# B&R Automation Studio project TD52 (part 53)

```c
  /* BusSelector: '<S111>/Bus Selector12' */
  rtb_rSCR_NOxControlWaiting = UDC_B.BusInput1.rSCR_NOxControlWaiting;

  /* UnitDelay: '<S111>/Unit Delay' */
  rtb_UnitDelay = UDC_DWork.UnitDelay_DSTATE;

  /* BusSelector: '<S113>/Bus Selector1' */
  for (i = 0; i < 5; i++) {
    rtb_rUrClKiOffs_y[i] = UDC_B.BusInput2.CLNOx.rUrClKpOffs_x[i];
  }

  for (i = 0; i < 5; i++) {
    rtb_rUrClKiOffs_x[i] = UDC_B.BusInput2.CLNOx.rUrClKpOffs_y[i];
  }

  /* End of BusSelector: '<S113>/Bus Selector1' */
  /* Dynamic Look-Up Table Block: '<S113>/Lookup Table Dynamic'
   * Input0  Data Type:  Floating Point real32_T
   * Input1  Data Type:  Floating Point real32_T
   * Input2  Data Type:  Floating Point real32_T
   * Output0 Data Type:  Floating Point real32_T
   * Lookup Method: Linear_Endpoint
   *
   */
  LookUp_real32_T_real32_T( &(rtb_LookupTableDynamic1), rtb_rUrClKiOffs_x,
    rtb_Switch6, rtb_rUrClKiOffs_y, 4U, inst);

  /* Sum: '<S113>/Add2' */
  rtb_etaVolConst = rtb_LookupTableDynamic1 + UDC_B.BusInput1.rSCR_NOxCtrl_Kp;

  /* BusSelector: '<S111>/Bus Selector14' */
  rtb_bRel_SCR_Dosing_n = UDC_B.BusInput.bRel_SCR_Dosing;

  /* Logic: '<S111>/Logical Operator5' */
  rtb_RelationalOperator2 = (UDC_B.BusInput.bSCR_UreaDosingUnit_Man &&
    UDC_B.BusInput1.bSCR_UreaFlowCtrl_Active);

  /* Outputs for Atomic SubSystem: '<S111>/TON' */
  UDC_TON(rtb_bRel_SCR_Dosing_n, rtb_rSCR_NOxControlWaiting, &UDC_B.TON_f,
          &UDC_DWork.TON_f, inst);

  /* End of Outputs for SubSystem: '<S111>/TON' */

  /* Outputs for Atomic SubSystem: '<Root>/SlipDetection' */
  /* Logic: '<S111>/Logical Operator' incorporates:
   *  BusCreator: '<S10>/Bus Creator'
   *  Logic: '<S111>/Logical Operator3'
   */
  rtb_LogicalOperator_p = (UDC_B.BusInput2.CLNOx.bUrClRes ||
    rtb_RelationalOperator2 || (!UDC_B.TON_f.LogicalOperator3) ||
    UDC_B.BusInput.bSCR_Man || UDC_B.BusInput.bSCR_NOxControl_Man ||
    rtb_RelationalOperator_mq || UDC_B.BusInput.bSCR_NH3SlipDetect_Blocked);

  /* End of Outputs for SubSystem: '<Root>/SlipDetection' */

  /* Logic: '<S111>/Logical Operator8' incorporates:
   *  BusCreator: '<S9>/Bus Creator'
   */
  rtb_RelationalOperator2 = (rtb_bFreezeCtr_j || rtb_LogicalOperator_p);

  /* Switch: '<S111>/Switch1' incorporates:
   *  Constant: '<S111>/Constant'
   *  Gain: '<S111>/Gain'
   *  MATLAB Function: '<S119>/MATLAB Function'
   *  Sum: '<S111>/Add7'
   */
  if (rtb_RelationalOperator2) {
    rtb_LookupTableDynamic1 = 0.0F;
  } else {
    /* Outputs for Atomic SubSystem: '<S9>/E21_NOxCatOutManager' */
    rtb_LookupTableDynamic1 = -(rtb_BusCreator_h_rNOx_SCR_CatOu - rNOx_Act);

    /* End of Outputs for SubSystem: '<S9>/E21_NOxCatOutManager' */
  }

  /* End of Switch: '<S111>/Switch1' */

  /* Gain: '<S112>/Gain' */
  rtb_LookupTableDynamic1 *= 0.001F;

  /* Product: '<S112>/Product' */
  rtb_Product_f = rtb_etaVolConst * rtb_LookupTableDynamic1;

  /* DiscreteIntegrator: '<S112>/Discrete-Time Integrator' */
  if (UDC_DWork.DiscreteTimeIntegrator_IC_LOADI != 0) {
    UDC_DWork.DiscreteTimeIntegrator_DSTATE_p = UDC_B.BusInput2.CLNOx.rUrClI0;
    if (UDC_DWork.DiscreteTimeIntegrator_DSTATE_p >= 3.402823466E+38F) {
      UDC_DWork.DiscreteTimeIntegrator_DSTATE_p = 3.402823466E+38F;
    } else {
      if (UDC_DWork.DiscreteTimeIntegrator_DSTATE_p <= -3.402823466E+38F) {
        UDC_DWork.DiscreteTimeIntegrator_DSTATE_p = -3.402823466E+38F;
      }
    }
  }

  if (rtb_LogicalOperator_p || (UDC_DWork.DiscreteTimeIntegrator_PrevRe_j != 0))
  {
    UDC_DWork.DiscreteTimeIntegrator_DSTATE_p = UDC_B.BusInput2.CLNOx.rUrClI0;
    if (UDC_DWork.DiscreteTimeIntegrator_DSTATE_p >= 3.402823466E+38F) {
      UDC_DWork.DiscreteTimeIntegrator_DSTATE_p = 3.402823466E+38F;
    } else {
      if (UDC_DWork.DiscreteTimeIntegrator_DSTATE_p <= -3.402823466E+38F) {
        UDC_DWork.DiscreteTimeIntegrator_DSTATE_p = -3.402823466E+38F;
      }
    }
  }

  if (UDC_DWork.DiscreteTimeIntegrator_DSTATE_p >= 3.402823466E+38F) {
    UDC_DWork.DiscreteTimeIntegrator_DSTATE_p = 3.402823466E+38F;
  } else {
    if (UDC_DWork.DiscreteTimeIntegrator_DSTATE_p <= -3.402823466E+38F) {
      UDC_DWork.DiscreteTimeIntegrator_DSTATE_p = -3.402823466E+38F;
    }
  }

  rtb_DiscreteTimeIntegrator = UDC_DWork.DiscreteTimeIntegrator_DSTATE_p;

  /* End of DiscreteIntegrator: '<S112>/Discrete-Time Integrator' */

  /* BusSelector: '<S113>/Bus Selector4' */
  for (i = 0; i < 5; i++) {
    rtb_rUrClKiOffs_x[i] = UDC_B.BusInput2.CLNOx.rUrClKdOffs_x[i];
  }

  for (i = 0; i < 5; i++) {
    rtb_rUrClKiOffs_y[i] = UDC_B.BusInput2.CLNOx.rUrClKdOffs_y[i];
  }

  /* End of BusSelector: '<S113>/Bus Selector4' */
  /* Dynamic Look-Up Table Block: '<S113>/Lookup Table Dynamic2'
   * Input0  Data Type:  Floating Point real32_T
   * Input1  Data Type:  Floating Point real32_T
   * Input2  Data Type:  Floating Point real32_T
   * Output0 Data Type:  Floating Point real32_T
   * Lookup Method: Linear_Endpoint
   *
   */
  LookUp_real32_T_real32_T( &(rtb_Switch2_mg), rtb_rUrClKiOffs_y, rtb_Switch6,
    rtb_rUrClKiOffs_x, 4U, inst);

  /* Product: '<S112>/Product2' incorporates:
   *  Sum: '<S113>/Add3'
   */
  rtb_etaVolConst = (rtb_Switch2_mg + UDC_B.BusInput1.rSCR_NOxCtrl_Kd) *
    rtb_LookupTableDynamic1;

  /* DiscreteIntegrator: '<S112>/Discrete-Time Integrator1' */
  if (UDC_DWork.DiscreteTimeIntegrator1_IC_LOAD != 0) {
    UDC_DWork.DiscreteTimeIntegrator1_DSTATE = UDC_B.BusInput2.CLNOx.rUrClD0;
    if (UDC_DWork.DiscreteTimeIntegrator1_DSTATE >= 3.402823466E+38F) {
      UDC_DWork.DiscreteTimeIntegrator1_DSTATE = 3.402823466E+38F;
    } else {
      if (UDC_DWork.DiscreteTimeIntegrator1_DSTATE <= -3.402823466E+38F) {
        UDC_DWork.DiscreteTimeIntegrator1_DSTATE = -3.402823466E+38F;
      }
    }
  }

  if (rtb_LogicalOperator_p || (UDC_DWork.DiscreteTimeIntegrator1_PrevRes != 0))
  {
    UDC_DWork.DiscreteTimeIntegrator1_DSTATE = UDC_B.BusInput2.CLNOx.rUrClD0;
    if (UDC_DWork.DiscreteTimeIntegrator1_DSTATE >= 3.402823466E+38F) {
      UDC_DWork.DiscreteTimeIntegrator1_DSTATE = 3.402823466E+38F;
    } else {
      if (UDC_DWork.DiscreteTimeIntegrator1_DSTATE <= -3.402823466E+38F) {
        UDC_DWork.DiscreteTimeIntegrator1_DSTATE = -3.402823466E+38F;
      }
    }
  }

  if (UDC_DWork.DiscreteTimeIntegrator1_DSTATE >= 3.402823466E+38F) {
    UDC_DWork.DiscreteTimeIntegrator1_DSTATE = 3.402823466E+38F;
  } else {
    if (UDC_DWork.DiscreteTimeIntegrator1_DSTATE <= -3.402823466E+38F) {
      UDC_DWork.DiscreteTimeIntegrator1_DSTATE = -3.402823466E+38F;
    }
  }

  rtb_Switch2_mg = UDC_DWork.DiscreteTimeIntegrator1_DSTATE;

  /* End of DiscreteIntegrator: '<S112>/Discrete-Time Integrator1' */

  /* Product: '<S112>/Product3' incorporates:
   *  Sum: '<S112>/Sum2'
   */
  rtb_Product3 = (rtb_etaVolConst - rtb_Switch2_mg) *
    UDC_B.BusInput2.CLNOx.rUrClN;

  /* Switch: '<S111>/Switch' incorporates:
   *  BusCreator: '<S9>/Bus Creator'
   *  Sum: '<S112>/Sum1'
   */
  if (!rtb_bFreezeCtr_j) {
    rtb_UnitDelay = (rtb_Product_f + rtb_DiscreteTimeIntegrator) + rtb_Product3;
  }

  /* End of Switch: '<S111>/Switch' */

  /* Switch: '<S114>/Switch2' incorporates:
   *  RelationalOperator: '<S114>/LowerRelop1'
   *  RelationalOperator: '<S114>/UpperRelop'
   *  Switch: '<S114>/Switch'
   */
  if (rtb_UnitDelay > UDC_B.BusInput1.rSCR_NOxCtrl_Ymax) {
    rtb_Switch2_m = UDC_B.BusInput1.rSCR_NOxCtrl_Ymax;
  } else if (rtb_UnitDelay < UDC_B.BusInput1.rSCR_NOxCtrl_Ymin) {
    /* Switch: '<S114>/Switch' */
    rtb_Switch2_m = UDC_B.BusInput1.rSCR_NOxCtrl_Ymin;
  } else {
    rtb_Switch2_m = rtb_UnitDelay;
  }

  /* End of Switch: '<S114>/Switch2' */

  /* Switch: '<S8>/Switch1' incorporates:
   *  Constant: '<S8>/const1'
   *  Switch: '<S8>/Switch7'
   */
  if (UDC_B.BusInput.bSCR_NOxControl_Man) {
    rtb_Switch_ah = UDC_B.BusInput.rFlow_SCR_UreaDosingUnit_spMan;
  } else if (UDC_B.BusInput.bRel_SCR_Dosing) {
    /* Switch: '<S8>/Switch7' incorporates:
     *  Sum: '<S8>/Add6'
     */
    rtb_Switch_ah = rtb_rFlow_SCR_UreaDosing_ffNH3C + rtb_Switch2_m;
  } else {
    rtb_Switch_ah = 0.0F;
  }

  /* End of Switch: '<S8>/Switch1' */

  /* Switch: '<S110>/Switch2' incorporates:
   *  Constant: '<S8>/const2'
   *  RelationalOperator: '<S110>/LowerRelop1'
   *  RelationalOperator: '<S110>/UpperRelop'
   *  Switch: '<S110>/Switch'
   */
  if (rtb_Switch_ah > UDC_B.BusInput1.rFlow_SCR_UreaDosingUnit_Hi) {
    rtb_Switch2_h = UDC_B.BusInput1.rFlow_SCR_UreaDosingUnit_Hi;
  } else if (rtb_Switch_ah < 0.0F) {
    /* Switch: '<S110>/Switch' incorporates:
     *  Constant: '<S8>/const2'
     */
    rtb_Switch2_h = 0.0F;
  } else {
    rtb_Switch2_h = rtb_Switch_ah;
  }

  /* End of Switch: '<S110>/Switch2' */

  /* If: '<S6>/If' incorporates:
   *  Constant: '<S84>/Constant'
   *  Constant: '<S84>/Constant1'
   *  Constant: '<S84>/Constant2'
   *  Constant: '<S84>/Constant7'
   *  Constant: '<S84>/Constant8'
   */
  if (UDC_B.BusInput1.bSCR_UreaDosingValve_Exist &&
      UDC_B.BusInput1.bSCR_UreaFlowCtrl_Active) {
    /* Outputs for IfAction SubSystem: '<S6>/UrValCntr' incorporates:
     *  ActionPort: '<S86>/Action Port'
     */
    /* Sum: '<S86>/Add2' */
    rtb_etaVolConst = UDC_B.BusInput2.CLVal.rUrValKpOffs +
      UDC_B.BusInput1.rSCR_UreaFlowCtrl_Kp;

    /* Switch: '<S86>/Switch1' incorporates:
     *  Constant: '<S86>/Constant'
     *  Sum: '<S86>/Add7'
     */
    if (UDC_B.BusInput.tFlow_SCR_UreaDosingOut.GoodQual) {
      rtb_Product_k = rtb_Switch2_h - UDC_B.BusInput.tFlow_SCR_UreaDosingOut.Ai;
    } else {
      rtb_Product_k = 0.0F;
    }

    /* End of Switch: '<S86>/Switch1' */

    /* Gain: '<S94>/Gain' */
    rtb_sampletime_c = 0.01F * rtb_Product_k;

    /* Product: '<S94>/Product' */
    rtb_Product_k = rtb_etaVolConst * rtb_sampletime_c;

    /* Logic: '<S86>/Logical Operator' incorporates:
     *  Logic: '<S86>/Logical Operator1'
     *  Logic: '<S86>/Logical Operator2'
     *  Logic: '<S86>/Logical Operator3'
     */
    rtb_LogicalOperator_g = (UDC_B.BusInput2.CLVal.bUrValRes ||
      (!UDC_B.BusInput1.bSCR_UreaDosingValve_Exist) ||
      (!UDC_B.BusInput.bRel_SCR_Dosing) ||
      (!UDC_B.BusInput1.bSCR_UreaFlowCtrl_Active) || UDC_B.BusInput.bSCR_Man ||
      UDC_B.BusInput.bSCR_UreaDosingUnit_Man);

    /* DiscreteIntegrator: '<S94>/Discrete-Time Integrator' */
    if (UDC_DWork.DiscreteTimeIntegrator_IC_LOA_f != 0) {
      UDC_DWork.DiscreteTimeIntegrator_DSTATE_e = UDC_B.BusInput2.CLVal.rUrValI0;
      if (UDC_DWork.DiscreteTimeIntegrator_DSTATE_e >= 3.402823466E+38F) {
        UDC_DWork.DiscreteTimeIntegrator_DSTATE_e = 3.402823466E+38F;
      } else {
        if (UDC_DWork.DiscreteTimeIntegrator_DSTATE_e <= -3.402823466E+38F) {
          UDC_DWork.DiscreteTimeIntegrator_DSTATE_e = -3.402823466E+38F;
        }
      }
    }

    if (rtb_LogicalOperator_g || (UDC_DWork.DiscreteTimeIntegrator_PrevRe_p != 0))
    {
      UDC_DWork.DiscreteTimeIntegrator_DSTATE_e = UDC_B.BusInput2.CLVal.rUrValI0;
      if (UDC_DWork.DiscreteTimeIntegrator_DSTATE_e >= 3.402823466E+38F) {
        UDC_DWork.DiscreteTimeIntegrator_DSTATE_e = 3.402823466E+38F;
      } else {
        if (UDC_DWork.DiscreteTimeIntegrator_DSTATE_e <= -3.402823466E+38F) {
          UDC_DWork.DiscreteTimeIntegrator_DSTATE_e = -3.402823466E+38F;
        }
      }
    }

    if (UDC_DWork.DiscreteTimeIntegrator_DSTATE_e >= 3.402823466E+38F) {
      UDC_DWork.DiscreteTimeIntegrator_DSTATE_e = 3.402823466E+38F;
    } else {
      if (UDC_DWork.DiscreteTimeIntegrator_DSTATE_e <= -3.402823466E+38F) {
        UDC_DWork.DiscreteTimeIntegrator_DSTATE_e = -3.402823466E+38F;
      }
    }

    rtb_DiscreteTimeIntegrator_p = UDC_DWork.DiscreteTimeIntegrator_DSTATE_e;

    /* Sum: '<S86>/Add6' */
    rtb_etaVolConst = UDC_B.BusInput2.CLVal.rUrValKdOffs +
      UDC_B.BusInput1.rSCR_UreaFlowCtrl_Kd;

    /* DiscreteIntegrator: '<S94>/Discrete-Time Integrator1' */
    if (UDC_DWork.DiscreteTimeIntegrator1_IC_LO_i != 0) {
      UDC_DWork.DiscreteTimeIntegrator1_DSTAT_b = UDC_B.BusInput2.CLVal.rUrValD0;
      if (UDC_DWork.DiscreteTimeIntegrator1_DSTAT_b >= 3.402823466E+38F) {
        UDC_DWork.DiscreteTimeIntegrator1_DSTAT_b = 3.402823466E+38F;
      } else {
        if (UDC_DWork.DiscreteTimeIntegrator1_DSTAT_b <= -3.402823466E+38F) {
          UDC_DWork.DiscreteTimeIntegrator1_DSTAT_b = -3.402823466E+38F;
        }
      }
    }

    if (rtb_LogicalOperator_g || (UDC_DWork.DiscreteTimeIntegrator1_PrevR_e != 0))
    {
      UDC_DWork.DiscreteTimeIntegrator1_DSTAT_b = UDC_B.BusInput2.CLVal.rUrValD0;
      if (UDC_DWork.DiscreteTimeIntegrator1_DSTAT_b >= 3.402823466E+38F) {
        UDC_DWork.DiscreteTimeIntegrator1_DSTAT_b = 3.402823466E+38F;
      } else {
        if (UDC_DWork.DiscreteTimeIntegrator1_DSTAT_b <= -3.402823466E+38F) {
          UDC_DWork.DiscreteTimeIntegrator1_DSTAT_b = -3.402823466E+38F;
        }
      }
    }

    if (UDC_DWork.DiscreteTimeIntegrator1_DSTAT_b >= 3.402823466E+38F) {
      UDC_DWork.DiscreteTimeIntegrator1_DSTAT_b = 3.402823466E+38F;
    } else {
      if (UDC_DWork.DiscreteTimeIntegrator1_DSTAT_b <= -3.402823466E+38F) {
        UDC_DWork.DiscreteTimeIntegrator1_DSTAT_b = -3.402823466E+38F;
      }
    }

    /* Product: '<S94>/Product3' incorporates:
     *  DiscreteIntegrator: '<S94>/Discrete-Time Integrator1'
     *  Product: '<S94>/Product2'
     *  Sum: '<S94>/Sum2'
     */
    rtb_Product3_i = (rtb_etaVolConst * rtb_sampletime_c -
                      UDC_DWork.DiscreteTimeIntegrator1_DSTAT_b) *
      UDC_B.BusInput2.CLVal.rUrValN;

    /* Switch: '<S86>/Switch' incorporates:
     *  DiscreteIntegrator: '<S94>/Discrete-Time Integrator'
     *  Sum: '<S94>/Sum1'
     *  UnitDelay: '<S86>/Unit Delay'
     */
    if (UDC_B.BusInput.tFlow_SCR_UreaDosingOut.GoodQual) {
      rtb_Switch2_kp = (rtb_Product_k +
                        UDC_DWork.DiscreteTimeIntegrator_DSTATE_e) +
        rtb_Product3_i;
    } else {
      rtb_Switch2_kp = UDC_DWork.UnitDelay_DSTATE_n;
    }

    /* End of Switch: '<S86>/Switch' */

    /* Switch: '<S95>/Switch2' incorporates:
     *  RelationalOperator: '<S95>/LowerRelop1'
     *  RelationalOperator: '<S95>/UpperRelop'
     *  Switch: '<S95>/Switch'
     */
    if (rtb_Switch2_kp > UDC_B.BusInput1.rSCR_UreaFlowCtrl_Ymax) {
      rtb_Switch2_p = UDC_B.BusInput1.rSCR_UreaFlowCtrl_Ymax;
    } else if (rtb_Switch2_kp < UDC_B.BusInput1.rSCR_UreaFlowCtrl_Ymin) {
      /* Switch: '<S95>/Switch' */
      rtb_Switch2_p = UDC_B.BusInput1.rSCR_UreaFlowCtrl_Ymin;
    } else {
      rtb_Switch2_p = rtb_Switch2_kp;
    }

    /* End of Switch: '<S95>/Switch2' */

    /* Abs: '<S93>/Abs' incorporates:
     *  BusSelector: '<S86>/Bus Selector1'
     */
    rtb_LookupTableDynamic_e = (real32_T)fabs
      (UDC_B.BusInput1.rFlow_SCR_UreaDosingValveCoeff);

    /* Switch: '<S93>/Switch' incorporates:
     *  BusSelector: '<S86>/Bus Selector1'
     *  Constant: '<S93>/Constant2'
     *  RelationalOperator: '<S93>/Relational Operator'
     */
    if (1.1920929E-7F >= rtb_LookupTableDynamic_e) {
      rtb_Switch_f = 1.1920929E-7F;
    } else {
      rtb_Switch_f = UDC_B.BusInput1.rFlow_SCR_UreaDosingValveCoeff;
    }

    /* End of Switch: '<S93>/Switch' */

    /* UnitDelay: '<S97>/Unit Delay' */
    rtb_LookupTableDynamic_e = UDC_DWork.UnitDelay_DSTATE_d;

    /* Switch: '<S97>/Switch' */
    if (UDC_B.BusInput.tDPr_UreaDosingUnit.GoodQual) {
      rtb_Switch_ld = UDC_B.BusInput.tDPr_UreaDosingUnit.Ai;
    } else {
      rtb_Switch_ld = rtb_LookupTableDynamic_e;
    }

    /* End of Switch: '<S97>/Switch' */

    /* BusSelector: '<S97>/Bus Selector2' */
    for (i = 0; i < 11; i++) {
      rtb_rUrValLinMap_x[i] = UDC_B.BusInput2.CLVal.rUrValLinMap_x[i];
    }

    for (i = 0; i < 11; i++) {
      rtb_rUrValLinMap_y[i] = UDC_B.BusInput2.CLVal.rUrValLinMap_y[i];
    }

    rtb_rTiFilt_DPrVlv = UDC_B.BusInput2.CLVal.rTiFilt_DPrVlv;

    /* End of BusSelector: '<S97>/Bus Selector2' */

    /* Outputs for Atomic SubSystem: '<S97>/Filter_DPr' */
    UDC_Filter(rtb_rTiFilt_DPrVlv, rtb_LogicalOperator_g, rtb_Switch_ld,
               &UDC_B.Filter_DPr, &UDC_DWork.Filter_DPr, inst);

    /* End of Outputs for SubSystem: '<S97>/Filter_DPr' */

    /* Product: '<S97>/Divide2' incorporates:
     *  Gain: '<S97>/Gain'
     */
    rtb_LookupTableDynamic_e = UDC_B.Filter_DPr.Switch / (0.001F * rtb_Switch);

    /* Saturate: '<S97>/Saturation' */
    if (rtb_LookupTableDynamic_e >= 1.0E+6F) {
      rtb_LookupTableDynamic_e = 1.0E+6F;
    } else {
      if (rtb_LookupTableDynamic_e <= 0.001F) {
        rtb_LookupTableDynamic_e = 0.001F;
      }
    }

    /* End of Saturate: '<S97>/Saturation' */

    /* Sqrt: '<S97>/Sqrt' */
    rtb_LookupTableDynamic_e = (real32_T)sqrt(rtb_LookupTableDynamic_e);

    /* Abs: '<S100>/Abs' */
    rtb_Switch_h = (real32_T)fabs(rtb_LookupTableDynamic_e);

    /* Switch: '<S100>/Switch' incorporates:
     *  Constant: '<S100>/Constant2'
     *  RelationalOperator: '<S100>/Relational Operator'
     */
    if (1.1920929E-7F >= rtb_Switch_h) {
      rtb_LookupTableDynamic_e = 1.1920929E-7F;
    }

    /* End of Switch: '<S100>/Switch' */

    /* Product: '<S97>/Divide1' */
    rtb_LookupTableDynamic_e = rtb_Switch2_h / rtb_Switch_f /
      rtb_LookupTableDynamic_e;

    /* Dynamic Look-Up Table Block: '<S97>/Lookup Table Dynamic'
     * Input0  Data Type:  Floating Point real32_T
     * Input1  Data Type:  Floating Point real32_T
     * Input2  Data Type:  Floating Point real32_T
     * Output0 Data Type:  Floating Point real32_T
     * Lookup Method: Linear_Endpoint
     *
     */
    LookUp_real32_T_real32_T( &(rtb_Switch_h), rtb_rUrValLinMap_y,
      rtb_LookupTableDynamic_e, rtb_rUrValLinMap_x, 10U, inst);

    /* Sum: '<S86>/Add3' */
    rtb_LookupTableDynamic_e = rtb_Switch_h + rtb_Switch2_p;

    /* Product: '<S86>/Divide1' incorporates:
     *  Sum: '<S86>/Add1'
     */
    rtb_etaVolConst = (rtb_Switch2_kp - rtb_Switch2_p) *
      UDC_B.BusInput2.CLVal.rUrValKaw;

    /* Product: '<S86>/Divide6' incorporates:
     *  Sum: '<S86>/Add10'
     */
    rtb_Gain1 = (rtb_LookupTableDynamic_e -
                 UDC_B.BusInput.rPos_SCR_UreaDosingValve) *
      UDC_B.BusInput2.CLVal.rUrValKawExt;

    /* Saturate: '<S86>/Saturation1' */
    if (rtb_LookupTableDynamic_e >= 1.0F) {
      rtb_Saturation1_f = 1.0F;
    } else if (rtb_LookupTableDynamic_e <= 0.0F) {
      rtb_Saturation1_f = 0.0F;
    } else {
      rtb_Saturation1_f = rtb_LookupTableDynamic_e;
    }

    /* End of Saturate: '<S86>/Saturation1' */

    /* Product: '<S86>/Divide2' incorporates:
     *  Sum: '<S86>/Add8'
     */
    rtb_UkYk1 = (rtb_LookupTableDynamic_e - rtb_Saturation1_f) *
      UDC_B.BusInput2.CLVal.rUrValKaw;

    /* Sum: '<S86>/Add4' */
    rtb_etaVolConst = (rtb_etaVolConst + rtb_Gain1) + rtb_UkYk1;

    /* Sum: '<S86>/Add5' */
    rtb_UkYk1 = UDC_B.BusInput2.CLVal.rUrValKiOffs +
      UDC_B.BusInput1.rSCR_UreaFlowCtrl_Ki;

    /* Switch: '<S96>/Switch2' incorporates:
     *  Gain: '<S86>/Gain3'
     *  RelationalOperator: '<S96>/LowerRelop1'
     *  RelationalOperator: '<S96>/UpperRelop'
     *  Switch: '<S96>/Switch'
     */
    if (rtb_etaVolConst > UDC_B.BusInput1.rFlow_SCR_UreaDosingUnit_Hi) {
      rtb_LookupTableDynamic_e = UDC_B.BusInput1.rFlow_SCR_UreaDosingUnit_Hi;
    } else if (rtb_etaVolConst < -UDC_B.BusInput1.rFlow_SCR_UreaDosingUnit_Hi) {
      /* Switch: '<S96>/Switch' incorporates:
       *  Gain: '<S86>/Gain3'
       */
      rtb_LookupTableDynamic_e = -UDC_B.BusInput1.rFlow_SCR_UreaDosingUnit_Hi;
    } else {
      /* Switch: '<S96>/Switch' */
      rtb_LookupTableDynamic_e = rtb_etaVolConst;
    }

    /* End of Switch: '<S96>/Switch2' */

    /* Gain: '<S86>/Gain2' */
    rtb_LookupTableDynamic_e = -rtb_LookupTableDynamic_e;

    /* Logic: '<S86>/Logical Operator4' */
    rtb_LogicalOperator1_b = !rtb_LogicalOperator_g;

    /* Sum: '<S94>/Add' */
    rtb_etaVolConst = rtb_sampletime_c + rtb_LookupTableDynamic_e;

    /* BusCreator: '<S94>/Bus Creator' */
    rtb_sampletime_c = rtb_LookupTableDynamic_e;

    /* SignalConversion: '<S86>/Signal Conversion' */
    UDC_B.Merge5[0] = rtb_Switch_h;

    /* SignalConversion: '<S86>/Signal Conversion1' */
    UDC_B.Merge5[1] = rtb_Saturation1_f;

    /* SignalConversion: '<S86>/Signal Conversion2' */
    UDC_B.Merge5[2] = rtb_Switch2_p;

    /* BusSelector: '<S98>/Bus Selector4' */
    for (i = 0; i < 11; i++) {
      rtb_rUrValLinMap_y[i] = UDC_B.BusInput2.CLVal.rUrValLinMap_y[i];
    }

    for (i = 0; i < 11; i++) {
      rtb_rUrValLinMap_x[i] = UDC_B.BusInput2.CLVal.rUrValLinMap_x[i];
    }

    rtb_rTiFilt_DPrVlv_b = UDC_B.BusInput2.CLVal.rTiFilt_DPrVlv;

    /* End of BusSelector: '<S98>/Bus Selector4' */

    /* UnitDelay: '<S98>/Unit Delay2' */
    rtb_Switch_h = UDC_DWork.UnitDelay2_DSTATE;

    /* Switch: '<S98>/Switch3' */
    if (UDC_B.BusInput.tDPr_UreaDosingUnit.GoodQual) {
      rtb_Switch3_l = UDC_B.BusInput.tDPr_UreaDosingUnit.Ai;
    } else {
      rtb_Switch3_l = rtb_Switch_h;
    }

    /* End of Switch: '<S98>/Switch3' */

    /* Outputs for Atomic SubSystem: '<S98>/Filter_DPr' */
    UDC_Filter(rtb_rTiFilt_DPrVlv_b, rtb_LogicalOperator_g, rtb_Switch3_l,
               &UDC_B.Filter_DPr_h, &UDC_DWork.Filter_DPr_h, inst);

    /* End of Outputs for SubSystem: '<S98>/Filter_DPr' */

    /* Product: '<S98>/Divide5' incorporates:
     *  Gain: '<S98>/Gain1'
     */
    rtb_Switch_h = UDC_B.Filter_DPr_h.Switch / (0.001F * rtb_Switch);

    /* Saturate: '<S98>/Saturation2' */
    if (rtb_Switch_h >= 1.0E+6F) {
      rtb_Switch_h = 1.0E+6F;
    } else {
      if (rtb_Switch_h <= 0.001F) {
        rtb_Switch_h = 0.001F;
      }
    }

    /* End of Saturate: '<S98>/Saturation2' */

    /* Sqrt: '<S98>/Sqrt1' */
    rtb_Switch_h = (real32_T)sqrt(rtb_Switch_h);

    /* Abs: '<S105>/Abs' */
    rtb_LookupTableDynamic_e = (real32_T)fabs(rtb_Switch_h);

    /* Switch: '<S105>/Switch' incorporates:
     *  Constant: '<S105>/Constant2'
     *  RelationalOperator: '<S105>/Relational Operator'
     */
    if (1.1920929E-7F >= rtb_LookupTableDynamic_e) {
      rtb_Switch_h = 1.1920929E-7F;
    }

    /* End of Switch: '<S105>/Switch' */
    /* Dynamic Look-Up Table Block: '<S98>/Lookup Table Dynamic'
     * Input0  Data Type:  Floating Point real32_T
     * Input1  Data Type:  Floating Point real32_T
     * Input2  Data Type:  Floating Point real32_T
     * Output0 Data Type:  Floating Point real32_T
     * Lookup Method: Linear_Endpoint
     *
     */
    LookUp_real32_T_real32_T( &(rtb_LookupTableDynamic_e), rtb_rUrValLinMap_x,
      rtb_Saturation1_f, rtb_rUrValLinMap_y, 10U, inst);

    /* Product: '<S98>/Divide4' */
    UDC_B.Merge5[3] = rtb_Switch_h * rtb_Switch_f * rtb_LookupTableDynamic_e;

    /* Update for DiscreteIntegrator: '<S94>/Discrete-Time Integrator' incorporates:
     *  Product: '<S94>/Product1'
     */
    UDC_DWork.DiscreteTimeIntegrator_IC_LOA_f = 0U;
    if (!rtb_LogicalOperator_g) {
      UDC_DWork.DiscreteTimeIntegrator_DSTATE_e += rtb_UkYk1 * rtb_etaVolConst *
        0.1F;
      if (UDC_DWork.DiscreteTimeIntegrator_DSTATE_e >= 3.402823466E+38F) {
        UDC_DWork.DiscreteTimeIntegrator_DSTATE_e = 3.402823466E+38F;
      } else {
        if (UDC_DWork.DiscreteTimeIntegrator_DSTATE_e <= -3.402823466E+38F) {
          UDC_DWork.DiscreteTimeIntegrator_DSTATE_e = -3.402823466E+38F;
        }
      }
    }

    if (rtb_LogicalOperator_g) {
      UDC_DWork.DiscreteTimeIntegrator_PrevRe_p = 1;
    } else {
      UDC_DWork.DiscreteTimeIntegrator_PrevRe_p = 0;
    }

    /* End of Update for DiscreteIntegrator: '<S94>/Discrete-Time Integrator' */

    /* Update for DiscreteIntegrator: '<S94>/Discrete-Time Integrator1' */
    UDC_DWork.DiscreteTimeIntegrator1_IC_LO_i = 0U;
    if (!rtb_LogicalOperator_g) {
      UDC_DWork.DiscreteTimeIntegrator1_DSTAT_b += 0.1F * rtb_Product3_i;
      if (UDC_DWork.DiscreteTimeIntegrator1_DSTAT_b >= 3.402823466E+38F) {
        UDC_DWork.DiscreteTimeIntegrator1_DSTAT_b = 3.402823466E+38F;
      } else {
        if (UDC_DWork.DiscreteTimeIntegrator1_DSTAT_b <= -3.402823466E+38F) {
          UDC_DWork.DiscreteTimeIntegrator1_DSTAT_b = -3.402823466E+38F;
        }
      }
    }

    if (rtb_LogicalOperator_g) {
      UDC_DWork.DiscreteTimeIntegrator1_PrevR_e = 1;
    } else {
      UDC_DWork.DiscreteTimeIntegrator1_PrevR_e = 0;
    }

    /* End of Update for DiscreteIntegrator: '<S94>/Discrete-Time Integrator1' */

    /* Update for UnitDelay: '<S86>/Unit Delay' */
    UDC_DWork.UnitDelay_DSTATE_n = rtb_Switch2_kp;

    /* Update for UnitDelay: '<S97>/Unit Delay' */
    UDC_DWork.UnitDelay_DSTATE_d = rtb_Switch_ld;

    /* Update for UnitDelay: '<S98>/Unit Delay2' */
    UDC_DWork.UnitDelay2_DSTATE = rtb_Switch3_l;

    /* End of Outputs for SubSystem: '<S6>/UrValCntr' */
  } else if (UDC_B.BusInput1.bSCR_UreaFlowCtrl_Active) {
    /* Outputs for IfAction SubSystem: '<S6>/UrPumpCntr' incorporates:
     *  ActionPort: '<S85>/Action Port'
     */
    /* BusSelector: '<S85>/Bus Selector2' */
    for (i = 0; i < 11; i++) {
      rtb_rUrPpCntrFFMap_x[i] = UDC_B.BusInput2.CLPp.rUrPpCntrFFMap_x[i];
    }

    for (i = 0; i < 11; i++) {
      rtb_rUrPpCntrFFMap_y[i] = UDC_B.BusInput2.CLPp.rUrPpCntrFFMap_y[i];
    }

    /* End of BusSelector: '<S85>/Bus Selector2' */

    /* Sum: '<S85>/Add2' */
    rtb_etaVolConst = UDC_B.BusInput2.CLPp.rUrPpKpOffs +
      UDC_B.BusInput1.rSCR_UreaFlowCtrl_Kp;

    /* Switch: '<S85>/Switch1' incorporates:
     *  Constant: '<S85>/Constant'
     *  Logic: '<S85>/Logical Operator6'
     *  Sum: '<S85>/Add7'
     */
    if (UDC_B.BusInput.tFlow_SCR_UreaDosingOut.GoodQual &&
        UDC_B.BusInput1.bFlow_SCR_UreaDosingOut_Exist) {
      rtb_Product_k = rtb_Switch2_h - UDC_B.BusInput.tFlow_SCR_UreaDosingOut.Ai;
    } else {
      rtb_Product_k = 0.0F;
    }

    /* End of Switch: '<S85>/Switch1' */

    /* Gain: '<S88>/Gain' */
    rtb_sampletime_c = 0.01F * rtb_Product_k;

    /* Product: '<S88>/Product' */
    rtb_Product_k = rtb_etaVolConst * rtb_sampletime_c;

    /* Logic: '<S85>/Logical Operator2' incorporates:
     *  Logic: '<S85>/Logical Operator1'
     *  Logic: '<S85>/Logical Operator3'
     *  Logic: '<S85>/Logical Operator5'
     */
    rtb_LogicalOperator2_j = (UDC_B.BusInput2.CLPp.bUrPpRes ||
      (!UDC_B.BusInput1.bSCR_UreaFlowCtrl_Active) ||
      (!UDC_B.BusInput.bRel_SCR_Dosing) || UDC_B.BusInput.bSCR_Man ||
      UDC_B.BusInput.bSCR_UreaDosingUnit_Man ||
      (!UDC_B.BusInput1.bFlow_SCR_UreaDosingOut_Exist));

    /* DiscreteIntegrator: '<S88>/Discrete-Time Integrator' */
    if (UDC_DWork.DiscreteTimeIntegrator_IC_LOA_e != 0) {
      UDC_DWork.DiscreteTimeIntegrator_DSTATE_d = UDC_B.BusInput2.CLPp.rUrPpI0;
      if (UDC_DWork.DiscreteTimeIntegrator_DSTATE_d >= 3.402823466E+38F) {
        UDC_DWork.DiscreteTimeIntegrator_DSTATE_d = 3.402823466E+38F;
      } else {
        if (UDC_DWork.DiscreteTimeIntegrator_DSTATE_d <= -3.402823466E+38F) {
          UDC_DWork.DiscreteTimeIntegrator_DSTATE_d = -3.402823466E+38F;
        }
      }
    }

    if (rtb_LogicalOperator2_j || (UDC_DWork.DiscreteTimeIntegrator_PrevR_j5 !=
         0)) {
      UDC_DWork.DiscreteTimeIntegrator_DSTATE_d = UDC_B.BusInput2.CLPp.rUrPpI0;
      if (UDC_DWork.DiscreteTimeIntegrator_DSTATE_d >= 3.402823466E+38F) {
        UDC_DWork.DiscreteTimeIntegrator_DSTATE_d = 3.402823466E+38F;
      } else {
        if (UDC_DWork.DiscreteTimeIntegrator_DSTATE_d <= -3.402823466E+38F) {
          UDC_DWork.DiscreteTimeIntegrator_DSTATE_d = -3.402823466E+38F;
        }
      }
    }

    if (UDC_DWork.DiscreteTimeIntegrator_DSTATE_d >= 3.402823466E+38F) {
      UDC_DWork.DiscreteTimeIntegrator_DSTATE_d = 3.402823466E+38F;
    } else {
      if (UDC_DWork.DiscreteTimeIntegrator_DSTATE_d <= -3.402823466E+38F) {
        UDC_DWork.DiscreteTimeIntegrator_DSTATE_d = -3.402823466E+38F;
      }
    }

    rtb_DiscreteTimeIntegrator_p = UDC_DWork.DiscreteTimeIntegrator_DSTATE_d;

    /* Sum: '<S85>/Add6' */
    rtb_etaVolConst = UDC_B.BusInput2.CLPp.rUrPpKdOffs +
      UDC_B.BusInput1.rSCR_UreaFlowCtrl_Kd;

    /* DiscreteIntegrator: '<S88>/Discrete-Time Integrator1' */
    if (UDC_DWork.DiscreteTimeIntegrator1_IC_LO_n != 0) {
      UDC_DWork.DiscreteTimeIntegrator1_DSTAT_l = UDC_B.BusInput2.CLPp.rUrPpD0;
      if (UDC_DWork.DiscreteTimeIntegrator1_DSTAT_l >= 3.402823466E+38F) {
        UDC_DWork.DiscreteTimeIntegrator1_DSTAT_l = 3.402823466E+38F;
      } else {
        if (UDC_DWork.DiscreteTimeIntegrator1_DSTAT_l <= -3.402823466E+38F) {
          UDC_DWork.DiscreteTimeIntegrator1_DSTAT_l = -3.402823466E+38F;
        }
      }
    }

    if (rtb_LogicalOperator2_j || (UDC_DWork.DiscreteTimeIntegrator1_PrevR_b !=
         0)) {
      UDC_DWork.DiscreteTimeIntegrator1_DSTAT_l = UDC_B.BusInput2.CLPp.rUrPpD0;
      if (UDC_DWork.DiscreteTimeIntegrator1_DSTAT_l >= 3.402823466E+38F) {
        UDC_DWork.DiscreteTimeIntegrator1_DSTAT_l = 3.402823466E+38F;
      } else {
        if (UDC_DWork.DiscreteTimeIntegrator1_DSTAT_l <= -3.402823466E+38F) {
          UDC_DWork.DiscreteTimeIntegrator1_DSTAT_l = -3.402823466E+38F;
        }
      }
    }

    if (UDC_DWork.DiscreteTimeIntegrator1_DSTAT_l >= 3.402823466E+38F) {
      UDC_DWork.DiscreteTimeIntegrator1_DSTAT_l = 3.402823466E+38F;
    } else {
      if (UDC_DWork.DiscreteTimeIntegrator1_DSTAT_l <= -3.402823466E+38F) {
        UDC_DWork.DiscreteTimeIntegrator1_DSTAT_l = -3.402823466E+38F;
      }
    }

    /* Product: '<S88>/Product3' incorporates:
     *  DiscreteIntegrator: '<S88>/Discrete-Time Integrator1'
     *  Product: '<S88>/Product2'
     *  Sum: '<S88>/Sum2'
     */
    rtb_Product3_i = (rtb_etaVolConst * rtb_sampletime_c -
                      UDC_DWork.DiscreteTimeIntegrator1_DSTAT_l) *
      UDC_B.BusInput2.CLPp.rUrPpN;

    /* Switch: '<S85>/Switch' incorporates:
     *  DiscreteIntegrator: '<S88>/Discrete-Time Integrator'
     *  Logic: '<S85>/Logical Operator7'
     *  Logic: '<S85>/Logical Operator8'
     *  Sum: '<S88>/Sum1'
     *  UnitDelay: '<S85>/Unit Delay'
     */
    if (UDC_B.BusInput.tFlow_SCR_UreaDosingOut.GoodQual ||
        (!UDC_B.BusInput1.bFlow_SCR_UreaDosingOut_Exist)) {
      rtb_Switch2_kp = (rtb_Product_k +
                        UDC_DWork.DiscreteTimeIntegrator_DSTATE_d) +
        rtb_Product3_i;
    } else {
      rtb_Switch2_kp = UDC_DWork.UnitDelay_DSTATE_j;
    }

    /* End of Switch: '<S85>/Switch' */

    /* Switch: '<S90>/Switch2' incorporates:
     *  RelationalOperator: '<S90>/LowerRelop1'
     *  RelationalOperator: '<S90>/UpperRelop'
     *  Switch: '<S90>/Switch'
     */
    if (rtb_Switch2_kp > UDC_B.BusInput1.rSCR_UreaFlowCtrl_Ymax) {
      rtb_Switch2_p = UDC_B.BusInput1.rSCR_UreaFlowCtrl_Ymax;
    } else if (rtb_Switch2_kp < UDC_B.BusInput1.rSCR_UreaFlowCtrl_Ymin) {
      /* Switch: '<S90>/Switch' */
      rtb_Switch2_p = UDC_B.BusInput1.rSCR_UreaFlowCtrl_Ymin;
    } else {
      rtb_Switch2_p = rtb_Switch2_kp;
    }

    /* End of Switch: '<S90>/Switch2' */

    /* Abs: '<S87>/Abs' */
    rtb_LookupTableDynamic_b = (real32_T)fabs
      (UDC_B.BusInput1.rFlow_SCR_UreaDosingUnit_Hi);

    /* Switch: '<S87>/Switch' incorporates:
     *  Constant: '<S87>/Constant2'
     *  RelationalOperator: '<S87>/Relational Operator'
     */
    if (1.1920929E-7F >= rtb_LookupTableDynamic_b) {
      rtb_LookupTableDynamic_b = 1.1920929E-7F;
    } else {
      rtb_LookupTableDynamic_b = UDC_B.BusInput1.rFlow_SCR_UreaDosingUnit_Hi;
    }

    /* End of Switch: '<S87>/Switch' */

    /* Product: '<S85>/Divide2' */
    rtb_LookupTableDynamic_b = 1.0F / rtb_LookupTableDynamic_b * rtb_Switch2_h;

    /* Dynamic Look-Up Table Block: '<S85>/Lookup Table Dynamic'
     * Input0  Data Type:  Floating Point real32_T
     * Input1  Data Type:  Floating Point real32_T
     * Input2  Data Type:  Floating Point real32_T
     * Output0 Data Type:  Floating Point real32_T
     * Lookup Method: Linear_Endpoint
     *
     */
    LookUp_real32_T_real32_T( &(rtb_LookupTableDynamic_f), rtb_rUrPpCntrFFMap_y,
      rtb_LookupTableDynamic_b, rtb_rUrPpCntrFFMap_x, 10U, inst);

    /* Sum: '<S85>/Add3' */
    rtb_LookupTableDynamic_b = rtb_LookupTableDynamic_f + rtb_Switch2_p;

    /* Product: '<S85>/Divide1' incorporates:
     *  Sum: '<S85>/Add1'
     */
    rtb_etaVolConst = (rtb_Switch2_kp - rtb_Switch2_p) *
      UDC_B.BusInput2.CLPp.rUrPpKaw;

    /* Product: '<S85>/Divide6' incorporates:
     *  Sum: '<S85>/Add10'
     */
    rtb_Gain1 = (rtb_LookupTableDynamic_b -
                 UDC_B.BusInput.rPc_SCR_UreaDosingPump) *
      UDC_B.BusInput2.CLPp.rUrPpKawExt;

    /* Saturate: '<S85>/Saturation1' */
    if (rtb_LookupTableDynamic_b >= 1.0F) {
      rtb_Saturation1 = 1.0F;
    } else if (rtb_LookupTableDynamic_b <= 0.0F) {
      rtb_Saturation1 = 0.0F;
    } else {
      rtb_Saturation1 = rtb_LookupTableDynamic_b;
    }

    /* End of Saturate: '<S85>/Saturation1' */

    /* Product: '<S85>/Divide3' incorporates:
     *  Sum: '<S85>/Add8'
     */
    rtb_UkYk1 = (rtb_LookupTableDynamic_b - rtb_Saturation1) *
      UDC_B.BusInput2.CLPp.rUrPpKaw;

    /* Sum: '<S85>/Add4' */
    rtb_etaVolConst = (rtb_etaVolConst + rtb_Gain1) + rtb_UkYk1;

    /* Sum: '<S85>/Add5' */
    rtb_UkYk1 = UDC_B.BusInput2.CLPp.rUrPpKiOffs +
      UDC_B.BusInput1.rSCR_UreaFlowCtrl_Ki;

    /* Switch: '<S91>/Switch2' incorporates:
     *  Gain: '<S85>/Gain2'
     *  RelationalOperator: '<S91>/LowerRelop1'
     *  RelationalOperator: '<S91>/UpperRelop'
     *  Switch: '<S91>/Switch'
     */
    if (rtb_etaVolConst > UDC_B.BusInput1.rFlow_SCR_UreaDosingUnit_Hi) {
      rtb_LookupTableDynamic_b = UDC_B.BusInput1.rFlow_SCR_UreaDosingUnit_Hi;
    } else if (rtb_etaVolConst < -UDC_B.BusInput1.rFlow_SCR_UreaDosingUnit_Hi) {
      /* Switch: '<S91>/Switch' incorporates:
       *  Gain: '<S85>/Gain2'
       */
      rtb_LookupTableDynamic_b = -UDC_B.BusInput1.rFlow_SCR_UreaDosingUnit_Hi;
    } else {
      /* Switch: '<S91>/Switch' */
      rtb_LookupTableDynamic_b = rtb_etaVolConst;
    }

    /* End of Switch: '<S91>/Switch2' */

    /* Gain: '<S85>/Gain1' */
    rtb_LookupTableDynamic_b = -rtb_LookupTableDynamic_b;

    /* Logic: '<S85>/Logical Operator4' */
    rtb_LogicalOperator1_b = !rtb_LogicalOperator2_j;

    /* Sum: '<S88>/Add' */
    rtb_etaVolConst = rtb_sampletime_c + rtb_LookupTableDynamic_b;

    /* BusCreator: '<S88>/Bus Creator' */
    rtb_sampletime_c = rtb_LookupTableDynamic_b;

    /* Dynamic Look-Up Table Block: '<S89>/Lookup Table Dynamic'
     * Input0  Data Type:  Floating Point real32_T
     * Input1  Data Type:  Floating Point real32_T
     * Input2  Data Type:  Floating Point real32_T
     * Output0 Data Type:  Floating Point real32_T
     * Lookup Method: Linear_Endpoint
     *
     */
    LookUp_real32_T_real32_T( &(rtb_LookupTableDynamic_b), rtb_rUrPpCntrFFMap_x,
      rtb_Saturation1, rtb_rUrPpCntrFFMap_y, 10U, inst);

    /* Product: '<S89>/Divide2' */
    UDC_B.Merge5[3] = rtb_LookupTableDynamic_b *
      UDC_B.BusInput1.rFlow_SCR_UreaDosingUnit_Hi;

    /* SignalConversion: '<S85>/Signal Conversion' */
    UDC_B.Merge5[0] = rtb_LookupTableDynamic_f;

    /* SignalConversion: '<S85>/Signal Conversion1' */
    UDC_B.Merge5[1] = rtb_Saturation1;

    /* SignalConversion: '<S85>/Signal Conversion2' */
    UDC_B.Merge5[2] = rtb_Switch2_p;

    /* Update for DiscreteIntegrator: '<S88>/Discrete-Time Integrator' incorporates:
     *  Product: '<S88>/Product1'
     */
    UDC_DWork.DiscreteTimeIntegrator_IC_LOA_e = 0U;
    if (!rtb_LogicalOperator2_j) {
      UDC_DWork.DiscreteTimeIntegrator_DSTATE_d += rtb_UkYk1 * rtb_etaVolConst *
        0.1F;
      if (UDC_DWork.DiscreteTimeIntegrator_DSTATE_d >= 3.402823466E+38F) {
        UDC_DWork.DiscreteTimeIntegrator_DSTATE_d = 3.402823466E+38F;
      } else {
        if (UDC_DWork.DiscreteTimeIntegrator_DSTATE_d <= -3.402823466E+38F) {
          UDC_DWork.DiscreteTimeIntegrator_DSTATE_d = -3.402823466E+38F;
        }
      }
    }

    if (rtb_LogicalOperator2_j) {
      UDC_DWork.DiscreteTimeIntegrator_PrevR_j5 = 1;
    } else {
      UDC_DWork.DiscreteTimeIntegrator_PrevR_j5 = 0;
    }

    /* End of Update for DiscreteIntegrator: '<S88>/Discrete-Time Integrator' */

    /* Update for DiscreteIntegrator: '<S88>/Discrete-Time Integrator1' */
    UDC_DWork.DiscreteTimeIntegrator1_IC_LO_n = 0U;
    if (!rtb_LogicalOperator2_j) {
      UDC_DWork.DiscreteTimeIntegrator1_DSTAT_l += 0.1F * rtb_Product3_i;
      if (UDC_DWork.DiscreteTimeIntegrator1_DSTAT_l >= 3.402823466E+38F) {
        UDC_DWork.DiscreteTimeIntegrator1_DSTAT_l = 3.402823466E+38F;
      } else {
        if (UDC_DWork.DiscreteTimeIntegrator1_DSTAT_l <= -3.402823466E+38F) {
          UDC_DWork.DiscreteTimeIntegrator1_DSTAT_l = -3.402823466E+38F;
        }
      }
    }

    if (rtb_LogicalOperator2_j) {
      UDC_DWork.DiscreteTimeIntegrator1_PrevR_b = 1;
    } else {
      UDC_DWork.DiscreteTimeIntegrator1_PrevR_b = 0;
    }

    /* End of Update for DiscreteIntegrator: '<S88>/Discrete-Time Integrator1' */

    /* Update for UnitDelay: '<S85>/Unit Delay' */
    UDC_DWork.UnitDelay_DSTATE_j = rtb_Switch2_kp;

    /* End of Outputs for SubSystem: '<S6>/UrPumpCntr' */
  } else {
    /* Outputs for IfAction SubSystem: '<S6>/Dummy' incorporates:
     *  ActionPort: '<S84>/Action Port'
     */
    UDC_B.Merge5[1] = 0.0F;
    UDC_B.Merge5[0] = 0.0F;
    UDC_B.Merge5[2] = 0.0F;
    UDC_B.Merge5[3] = 0.0F;
    rtb_LogicalOperator1_b = FALSE;

    /* BusCreator: '<S84>/Bus Creator' incorporates:
     *  Constant: '<S84>/Constant'
     *  Constant: '<S84>/Constant1'
     *  Constant: '<S84>/Constant2'
     *  Constant: '<S84>/Constant3'
     *  Constant: '<S84>/Constant4'
     *  Constant: '<S84>/Constant5'
     *  Constant: '<S84>/Constant6'
     *  Constant: '<S84>/Constant7'
     *  Constant: '<S84>/Constant8'
     */
    rtb_Product_k = 0.0F;
    rtb_DiscreteTimeIntegrator_p = 0.0F;
    rtb_Product3_i = 0.0F;
    rtb_sampletime_c = 0.0F;

    /* End of Outputs for SubSystem: '<S6>/Dummy' */
  }

  /* End of If: '<S6>/If' */

  /* BusCreator: '<Root>/Bus Creator1' incorporates:
   *  BusCreator: '<S10>/Bus Creator'
   *  BusCreator: '<S9>/Bus Creator'
   *  Logic: '<S111>/Logical Operator4'
   *  MATLAB Function: '<S119>/MATLAB Function'
   */
  UDC_Y.OutUDbus.rFlow_SCR_UreaDosingUnit_sp = rtb_Switch2_h;
  UDC_Y.OutUDbus.rFlow_SCR_NOxCtrl_Y = rtb_Switch2_m;
  UDC_Y.OutUDbus.bSCR_NOxCtrl_Act = !rtb_RelationalOperator2;

  /* Outputs for Atomic SubSystem: '<S9>/E21_NOxCatOutManager' */
  UDC_Y.OutUDbus.rNOx_SCR_NOxCtrl_act = rNOx_Act;

  /* End of Outputs for SubSystem: '<S9>/E21_NOxCatOutManager' */
  UDC_Y.OutUDbus.rNOx_SCR_CatOut_Set = rtb_BusCreator_h_rNOx_SCR_CatOu;
  UDC_Y.OutUDbus.bSCR_EngineSteadyState = rtb_LogicalOperator1_f;
  UDC_Y.OutUDbus.rPc_SCR_UreaDosingUnit_sp = UDC_B.Merge5[1];
  UDC_Y.OutUDbus.rPc_SCR_UreaDosingUnit_ff = UDC_B.Merge5[0];
  UDC_Y.OutUDbus.rPc_SCR_UreaFlowCtrl_Y = UDC_B.Merge5[2];
  UDC_Y.OutUDbus.bSCR_UreaFlowCtrl_Act = rtb_LogicalOperator1_b;
  UDC_Y.OutUDbus.rFlow_SCR_UreaDosingValve_Calc = UDC_B.Merge5[3];
  UDC_Y.OutUDbus.bSCR_NH3SlipDetected = rtb_LogicalOperator1_o;

  /* Outputs for Atomic SubSystem: '<Root>/SlipDetection' */
  UDC_Y.OutUDbus.bSCR_NH3SlipInterrupt = rtb_bSCR_NH3SlipInterrupt_k;

  /* End of Outputs for SubSystem: '<Root>/SlipDetection' */
  UDC_Y.OutUDbus.bSCR_EMValve1_SGbOxi_Dem = rtb_BusCreator_h3_bSCR_EMValve1;
  UDC_Y.OutUDbus.rFlow_SCR_UreaDosingUnit_ff = rtb_rFlow_SCR_UreaDosingUnit_ff;
  UDC_Y.OutUDbus.rUreaGain_Adj = rtb_DifferenceInputs2;
  UDC_Y.OutUDbus.rFlow_SCR_UreaDosing_ffNH3Cor = rtb_rFlow_SCR_UreaDosing_ffNH3C;

  /* Switch: '<S111>/Switch2' incorporates:
   *  BusCreator: '<S9>/Bus Creator'
   *  Constant: '<S111>/Constant1'
   *  Gain: '<S111>/Gain2'
   *  Sum: '<S111>/Add1'
   */
  if (rtb_bFreezeCtr_j) {
    rtb_etaVolConst = 0.0F;
  } else {
    /* Product: '<S111>/Divide6' incorporates:
     *  Sum: '<S111>/Add10'
     *  UnitDelay: '<S8>/Unit Delay'
     */
    rtb_UkYk1 = (UDC_DWork.UnitDelay_DSTATE_g -
                 UDC_B.BusInput.tFlow_SCR_UreaDosingOut.Ai) *
      UDC_B.BusInput2.CLNOx.rUrClKawExt;

    /* Product: '<S111>/Divide1' incorporates:
     *  Sum: '<S8>/Sum'
     */
    rtb_Gain1 = (rtb_Switch_ah - rtb_Switch2_h) * UDC_B.BusInput2.CLNOx.rUrClKaw;

    /* Product: '<S111>/Divide5' incorporates:
     *  Sum: '<S111>/Add9'
     */
    rtb_etaVolConst = (rtb_UnitDelay - rtb_Switch2_m) *
      UDC_B.BusInput2.CLNOx.rUrClKaw;
    rtb_etaVolConst = -((rtb_etaVolConst + rtb_Gain1) + rtb_UkYk1);
  }

  /* End of Switch: '<S111>/Switch2' */

  /* Switch: '<S115>/Switch2' incorporates:
   *  Gain: '<S111>/Gain1'
   *  RelationalOperator: '<S115>/LowerRelop1'
   *  RelationalOperator: '<S115>/UpperRelop'
   *  Switch: '<S115>/Switch'
   */
  if (rtb_etaVolConst > UDC_B.BusInput1.rNOx_SCR_CatOut_Hi) {
    rtb_Switch2_mg = UDC_B.BusInput1.rNOx_SCR_CatOut_Hi;
  } else if (rtb_etaVolConst < -UDC_B.BusInput1.rNOx_SCR_CatOut_Hi) {
    /* Switch: '<S115>/Switch' incorporates:
     *  Gain: '<S111>/Gain1'
     */
    rtb_Switch2_mg = -UDC_B.BusInput1.rNOx_SCR_CatOut_Hi;
  } else {
    /* Switch: '<S115>/Switch' */
    rtb_Switch2_mg = rtb_etaVolConst;
  }

  /* End of Switch: '<S115>/Switch2' */

  /* RelationalOperator: '<S111>/Relational Operator' */
  rtb_RelationalOperator2 = (rtb_UnitDelay >= UDC_B.BusInput1.rSCR_NOxCtrl_Ymax);

  /* BusCreator: '<Root>/Bus Creator' incorporates:
   *  BusCreator: '<S10>/Bus Creator'
   *  BusCreator: '<S111>/Bus Creator'
   *  BusCreator: '<S112>/Bus Creator'
   *  BusCreator: '<S5>/Bus Creator'
   *  BusCreator: '<S9>/Bus Creator'
   *  MATLAB Function: '<S119>/MATLAB Function'
   */
  UDC_Y.DebugUDbus.SM.rNOx_SCR_CatOut_Set = rtb_BusCreator_h_rNOx_SCR_CatOu;

  /* Outputs for Atomic SubSystem: '<S9>/E21_NOxCatOutManager' */
  UDC_Y.DebugUDbus.SM.rNOx_EMLineCatOut = rNOx_EMLineCatOut;
  UDC_Y.DebugUDbus.SM.bEMLineCatOut_GQ = bEMLineCatOut_GQ;
  UDC_Y.DebugUDbus.SM.rNOx_EMLineOxiIn = rNOx_EMLineOxiIn;
  UDC_Y.DebugUDbus.SM.bEMLineOxiIn_GQ = bEMLineOxiIn_GQ;
  UDC_Y.DebugUDbus.SM.rNOx_SCR_NOxCtrl_act = rNOx_Act;

  /* End of Outputs for SubSystem: '<S9>/E21_NOxCatOutManager' */
  UDC_Y.DebugUDbus.SM.bFreezeCtr = rtb_bFreezeCtr_j;
  UDC_Y.DebugUDbus.SM.rNOx_CatOutCor = rtb_rNOx_CatOutCor_k;
  UDC_Y.DebugUDbus.SM.bNOx_CatOutCor = rtb_bNOx_CatOutCor_n;
  UDC_Y.DebugUDbus.SM.rNOxEngOutCor = rtb_rNOxEngOutCor_e;
  UDC_Y.DebugUDbus.SM.bSCR_EngineSteadyState = rtb_LogicalOperator1_f;
  UDC_Y.DebugUDbus.SM.rTSCRAvg = rtb_BusCreator_h_rTSCRAvg;
  UDC_Y.DebugUDbus.FF.rSV = rtb_rSV;
  UDC_Y.DebugUDbus.FF.rMdot_exh = rtb_rMdot_exh;
  UDC_Y.DebugUDbus.FF.rTSCRAvgEst = rtb_Divide_h;
  UDC_Y.DebugUDbus.FF.rTSCRAvgAr = rtb_rTSCRAvg;
  UDC_Y.DebugUDbus.FF.rTSCRAvg = rtb_Switch6;
  UDC_Y.DebugUDbus.FF.rNH3StDMaxAvgEst = rtb_Divide1_o;
  UDC_Y.DebugUDbus.FF.rNH3StDMaxAr = rtb_LookupTableDynamic;
  UDC_Y.DebugUDbus.FF.rNH3StDEst = rtb_DiscreteTimeIntegrator_b;
  UDC_Y.DebugUDbus.FF.rNH3InFFSS = rtb_Divide2_h;
  UDC_Y.DebugUDbus.FF.rNH3InFF = rtb_Switch_kk;
  UDC_Y.DebugUDbus.FF.rdeltaNH3InTr = rtb_Switch_jg;
  UDC_Y.DebugUDbus.FF.rdeltaNH3InTr2 = rtb_Switch_ky;
  UDC_Y.DebugUDbus.FF.rNH3StDEst2 = rtb_Saturation_m;
  UDC_Y.DebugUDbus.FF.iIdxFFOut = rtb_iIdxFFOut;
  UDC_Y.DebugUDbus.FF.rFlowUreaFF_LT = rtb_rFlowUreaFF_LT;
  UDC_Y.DebugUDbus.FF.rFlowUreaFF_NOx = rtb_rFlowUreaFF_NOx_i;
  UDC_Y.DebugUDbus.FF.rFlowUreaFF_Map = rtb_rFlowUreaFF_Map;
  UDC_Y.DebugUDbus.FF.rFlowUreaFF_NH3 = rtb_rFlowUreaFF_NH3;
  UDC_Y.DebugUDbus.FF.rDensUrea = rtb_Switch;
  UDC_Y.DebugUDbus.Slip.bSCR_NH3SlipDetected = rtb_LogicalOperator1_o;
  UDC_Y.DebugUDbus.Slip.rUrCorFactSlip = rtb_BusCreator_h3_rUrCorFactSli;

  /* Outputs for Atomic SubSystem: '<Root>/SlipDetection' */
  UDC_Y.DebugUDbus.Slip.bFreezeCtrl = rtb_RelationalOperator_mq;
  UDC_Y.DebugUDbus.Slip.bSCR_NH3SlipInterrupt = rtb_bSCR_NH3SlipInterrupt_k;
  UDC_Y.DebugUDbus.Slip.bNH3SlipCtrlEna = rtb_bNH3SlipCtrlEna;

  /* End of Outputs for SubSystem: '<Root>/SlipDetection' */
  UDC_Y.DebugUDbus.Slip.bSCR_EMValve1_SGbOxi_Dem =
    rtb_BusCreator_h3_bSCR_EMValve1;
  UDC_Y.DebugUDbus.CLNOx.up = rtb_Product_f;
  UDC_Y.DebugUDbus.CLNOx.ui = rtb_DiscreteTimeIntegrator;
  UDC_Y.DebugUDbus.CLNOx.ud = rtb_Product3;
  UDC_Y.DebugUDbus.CLNOx.aw = rtb_Switch2_mg;
  UDC_Y.DebugUDbus.CLNOx.bFreeze = rtb_bFreezeCtr_j;
  UDC_Y.DebugUDbus.CLNOx.bSatUpLim = rtb_RelationalOperator2;
  UDC_Y.DebugUDbus.CLFlow.up = rtb_Product_k;
  UDC_Y.DebugUDbus.CLFlow.ui = rtb_DiscreteTimeIntegrator_p;
  UDC_Y.DebugUDbus.CLFlow.ud = rtb_Product3_i;
  UDC_Y.DebugUDbus.CLFlow.aw = rtb_sampletime_c;

  /* S-Function (bur_bus_out): '<Root>/Bus Output' */
  inst->dbg = UDC_Y.DebugUDbus;

  /* S-Function (bur_bus_out): '<Root>/Bus Output1' */
  inst->Out = UDC_Y.OutUDbus;

  /* BusSelector: '<Root>/Bus Selector10' incorporates:
   *  BusCreator: '<S111>/Bus Creator'
   */
  rtb_bSatUpLim_k = rtb_RelationalOperator2;

  /* Product: '<S28>/Divide3' */
  rtb_sampletime_c = rtb_Divide5 * UDC_B.BusInput2.FF.rNH3InTrGainA;

  /* Product: '<S29>/Divide5' */
  rtb_Switch2_kp = UDC_B.BusInput2.FF.rGainDeload * rtb_Saturation_m;

  /* Switch: '<S29>/Switch2' incorporates:
   *  Constant: '<S29>/I4'
   *  Constant: '<S29>/I5'
   */
  if (UDC_B.BusInput.bRel_SCR_Dosing) {
    i = 1;
  } else {
    i = 0;
  }

  /* End of Switch: '<S29>/Switch2' */

  /* Switch: '<S29>/Switch' incorporates:
   *  Constant: '<S29>/I1'
   *  Constant: '<S29>/I2'
   */
  if (UDC_B.BusInput.bOpModeStop) {
    tmp = 0;
  } else {
    tmp = 1;
  }

  /* End of Switch: '<S29>/Switch' */

  /* Product: '<S29>/Divide2' incorporates:
   *  BusCreator: '<S9>/Bus Creator'
   *  Product: '<S29>/Divide3'
   *  Product: '<S29>/Divide4'
   *  Sum: '<S29>/Add1'
   *  Sum: '<S29>/Add2'
   */
  rtb_Switch_f = ((real32_T)i * rtb_Switch_kk - (rtb_rNOxEngOutCor_e -
    rtb_rNOx_CatOutCor_k)) * (real32_T)tmp * UDC_B.BusInput2.FF.rNH3InTrGainC;

  /* BusSelector: '<S15>/Bus Selector5' */
  rtb_Ai_j0 = UDC_B.BusInput.tFlow_SCR_UreaDosingOut.Ai;

  /* BusSelector: '<S65>/Bus Selector3' */
  rtb_rTiConstAvgOn = UDC_B.BusInput2.FF.rTiConstAvgOn;
  rtb_rTiConstAvgOff = UDC_B.BusInput2.FF.rTiConstAvgOff;

  /* RelationalOperator: '<S65>/Relational Operator' */
  rtb_RelationalOperator2 = (UDC_B.BusInput.rP_Act_Norm_Filt >=
    UDC_B.BusInput2.FF.rPnorm_Thresh);

  /* Logic: '<S65>/Logical Operator' incorporates:
   *  BusCreator: '<S9>/Bus Creator'
   *  Logic: '<S65>/Logical Operator2'
   *  Logic: '<S65>/Logical Operator3'
   *  UnitDelay: '<S65>/Unit Delay4'
   */
  rtb_LogicalOperator_b = ((!UDC_B.BusInput.bSCR_Man) &&
    UDC_B.BusInput.bRel_SCR_Dosing &&
    UDC_B.BusInput.tFlow_SCR_UreaDosingOut.GoodQual && rtb_RelationalOperator2 &&
    rtb_LogicalOperator1_f && UDC_B.BusInput1.bSCR_Active &&
    UDC_B.BusInput1.bSCR_UreaNFlowAutoCorr_Active &&
    (!UDC_DWork.UnitDelay4_DSTATE_j));

  /* Logic: '<S65>/Logical Operator1' */
  rtb_LogicalOperator1_n = !rtb_LogicalOperator_b;

  /* Outputs for Atomic SubSystem: '<S15>/Filter' */
  UDC_Filter(rtb_rTiFiltUreaFFAdjust, rtb_LogicalOperator1_n, rtb_Ai_j0,
             &UDC_B.Filter_o, &UDC_DWork.Filter_o, inst);

  /* End of Outputs for SubSystem: '<S15>/Filter' */

  /* Outputs for Atomic SubSystem: '<S15>/Filter1' */
  UDC_Filter(rtb_rTiFiltUreaFFAdjust, rtb_LogicalOperator1_n,
             rtb_rFlow_SCR_UreaDosingUnit_ff, &UDC_B.Filter1, &UDC_DWork.Filter1, inst);

  /* End of Outputs for SubSystem: '<S15>/Filter1' */

  /* Outputs for Atomic SubSystem: '<S65>/TON' */
  UDC_TON(rtb_LogicalOperator_b, rtb_rTiConstAvgOn, &UDC_B.TON_j,
          &UDC_DWork.TON_j, inst);

  /* End of Outputs for SubSystem: '<S65>/TON' */

  /* Switch: '<S15>/Switch' */
  if (UDC_B.TON_j.LogicalOperator3) {
    /* Switch: '<S61>/Switch' incorporates:
     *  Abs: '<S61>/Abs'
     *  RelationalOperator: '<S61>/Relational Operator'
     */
    if (0.001F >= (real32_T)fabs(UDC_B.Filter1.Switch)) {
      rtb_Product_k = 0.001F;
    } else {
      rtb_Product_k = UDC_B.Filter1.Switch;
    }

    /* End of Switch: '<S61>/Switch' */

    /* Sum: '<S15>/Add1' incorporates:
     *  Constant: '<S15>/Constant15'
     *  Product: '<S15>/Divide2'
     *  Product: '<S15>/Product1'
     *  Sum: '<S15>/Add4'
     *  Sum: '<S15>/Add5'
     */
    rtb_etaVolConst = (UDC_B.Filter_o.Switch / rtb_Product_k - 1.0F) *
      (UDC_B.BusInput1.rCF_SCR_UreaNFlowGain + rtb_Switch2_l) + rtb_Switch2_l;

    /* RelationalOperator: '<S64>/LowerRelop1' */
    rtb_RelationalOperator2 = (rtb_etaVolConst >
      UDC_B.BusInput2.FF.rUreaGainDeltaLim);

    /* Switch: '<S64>/Switch2' */
    if (rtb_RelationalOperator2) {
      rtb_Switch2_l = UDC_B.BusInput2.FF.rUreaGainDeltaLim;
    } else {
      /* Gain: '<S15>/Gain2' */
      rtb_Gain1 = -UDC_B.BusInput2.FF.rUreaGainDeltaLim;

      /* Switch: '<S64>/Switch' incorporates:
       *  RelationalOperator: '<S64>/UpperRelop'
       */
      if (rtb_etaVolConst < rtb_Gain1) {
        rtb_Switch2_l = rtb_Gain1;
      } else {
        rtb_Switch2_l = rtb_etaVolConst;
      }

      /* End of Switch: '<S64>/Switch' */
    }

    /* End of Switch: '<S64>/Switch2' */
  }

  /* End of Switch: '<S15>/Switch' */

  /* Outputs for Atomic SubSystem: '<S65>/TP' */
  UDC_TP(UDC_B.TON_j.LogicalOperator3, rtb_rTiConstAvgOff, &UDC_B.TP,
         &UDC_DWork.TP, inst);

  /* End of Outputs for SubSystem: '<S65>/TP' */

  /* Sum: '<S112>/Add' */
  rtb_etaVolConst = rtb_LookupTableDynamic1 + rtb_Switch2_mg;

  /* BusSelector: '<S113>/Bus Selector3' */
  for (i = 0; i < 5; i++) {
    rtb_rUrClKiOffs_x[i] = UDC_B.BusInput2.CLNOx.rUrClKiOffs_x[i];
  }

  for (i = 0; i < 5; i++) {
    rtb_rUrClKiOffs_y[i] = UDC_B.BusInput2.CLNOx.rUrClKiOffs_y[i];
  }

  /* End of BusSelector: '<S113>/Bus Selector3' */
  /* Dynamic Look-Up Table Block: '<S113>/Lookup Table Dynamic1'
   * Input0  Data Type:  Floating Point real32_T
   * Input1  Data Type:  Floating Point real32_T
   * Input2  Data Type:  Floating Point real32_T
   * Output0 Data Type:  Floating Point real32_T
   * Lookup Method: Linear_Endpoint
   *
   */
  LookUp_real32_T_real32_T( &(rtb_LookupTableDynamic1), rtb_rUrClKiOffs_y,
    rtb_Switch6, rtb_rUrClKiOffs_x, 4U, inst);

  /* Sum: '<S113>/Add1' */
  rtb_Gain1 = rtb_LookupTableDynamic1 + UDC_B.BusInput1.rSCR_NOxCtrl_Ki;

  /* UnitDelay: '<S7>/Unit Delay' */
  UDC_B.UnitDelay = UDC_DWork.UnitDelay_DSTATE_c;

  /* S-Function (bur_out): '<Root>/Output' */
  inst->Version = UDC_B.UnitDelay;

  /* Update for Delay: '<S15>/Delay' */
  UDC_DWork.Delay_DSTATE = rtb_Switch2_l;

  /* Update for Delay: '<S66>/Delay' */
  UDC_DWork.icLoad = 0U;
  UDC_DWork.Delay_DSTATE_d = rtb_DifferenceInputs2;

  /* Update for Atomic SubSystem: '<Root>/SlipDetection' */
  /* Update for UnitDelay: '<S10>/Unit Delay' */
  UDC_DWork.UnitDelay_DSTATE_l = rtb_Compare_l;

  /* Update for UnitDelay: '<S142>/Delay Input1' */
  UDC_DWork.DelayInput1_DSTATE = rtb_UnitDelay_h;

  /* Update for UnitDelay: '<S141>/Unit Delay' */
  UDC_DWork.UnitDelay_DSTATE_dg = rtb_Compare_l;

  /* Update for UnitDelay: '<S138>/Unit Delay2' */
  UDC_DWork.UnitDelay2_DSTATE_f = rtb_LogicalOperator8;

  /* Update for UnitDelay: '<S10>/Unit Delay2' */
  UDC_DWork.UnitDelay2_DSTATE_i = rtb_bSatUpLim_k;

  /* Update for UnitDelay: '<S139>/Unit Delay4' */
  UDC_DWork.UnitDelay4_DSTATE = rtb_Switch4;

  /* Update for Memory: '<S156>/Memory' */
  UDC_DWork.Memory_PreviousInput = rtb_Logic[0];

  /* Update for UnitDelay: '<S198>/Delay Input1' */
  UDC_DWork.DelayInput1_DSTATE_m = rtb_Compare;

  /* Update for Delay: '<S202>/Delay' */
  UDC_DWork.icLoad_g = 0U;
  UDC_DWork.Delay_DSTATE_k = rtb_DifferenceInputs2_i;

  /* Update for Delay: '<S203>/Delay' */
  UDC_DWork.icLoad_e = 0U;
  UDC_DWork.Delay_DSTATE_h = rtb_DifferenceInputs2_a;

  /* Update for Memory: '<S200>/Memory' */
  UDC_DWork.Memory_PreviousInput_k = rtb_Logic_k[0];

  /* End of Update for SubSystem: '<Root>/SlipDetection' */

  /* Update for DiscreteIntegrator: '<S28>/Discrete-Time Integrator' */
  if (!rtb_bNH3StDRes) {
    UDC_DWork.DiscreteTimeIntegrator_DSTATE += 0.1F * rtb_sampletime_c;
  }

  if (rtb_bNH3StDRes) {
    UDC_DWork.DiscreteTimeIntegrator_PrevRese = 1;
  } else {
    UDC_DWork.DiscreteTimeIntegrator_PrevRese = 0;
  }

  /* End of Update for DiscreteIntegrator: '<S28>/Discrete-Time Integrator' */

  /* Update for DiscreteIntegrator: '<S29>/Discrete-Time Integrator' incorporates:
   *  Gain: '<S29>/Gain'
   *  Sum: '<S29>/Add4'
   *  Sum: '<S29>/Add5'
   *  Sum: '<S29>/Add6'
   */
  if (!rtb_bNH3StDRes2) {
    UDC_DWork.DiscreteTimeIntegrator_DSTATE_i += ((rtb_Switch_f - rtb_Switch2_kp)
      - (rtb_DiscreteTimeIntegrator_a - rtb_Saturation_m) * 100.0F) * 0.1F;
  }

  if (rtb_bNH3StDRes2) {
    UDC_DWork.DiscreteTimeIntegrator_PrevRe_k = 1;
  } else {
    UDC_DWork.DiscreteTimeIntegrator_PrevRe_k = 0;
  }

  /* End of Update for DiscreteIntegrator: '<S29>/Discrete-Time Integrator' */

  /* Update for Delay: '<S16>/Variable Integer Delay' */
  for (i = 0; i < 999; i++) {
    UDC_DWork.VariableIntegerDelay_DSTATE[i] =
      UDC_DWork.VariableIntegerDelay_DSTATE[i + 1];
  }

  UDC_DWork.VariableIntegerDelay_DSTATE[999] = rtb_Divide1_m;

  /* End of Update for Delay: '<S16>/Variable Integer Delay' */

  /* Update for UnitDelay: '<S111>/Unit Delay' */
  UDC_DWork.UnitDelay_DSTATE = rtb_UnitDelay;

  /* Update for DiscreteIntegrator: '<S112>/Discrete-Time Integrator' incorporates:
   *  Product: '<S112>/Product1'
   */
  UDC_DWork.DiscreteTimeIntegrator_IC_LOADI = 0U;
  if (!rtb_LogicalOperator_p) {
    UDC_DWork.DiscreteTimeIntegrator_DSTATE_p += rtb_Gain1 * rtb_etaVolConst *
      0.1F;
    if (UDC_DWork.DiscreteTimeIntegrator_DSTATE_p >= 3.402823466E+38F) {
      UDC_DWork.DiscreteTimeIntegrator_DSTATE_p = 3.402823466E+38F;
    } else {
      if (UDC_DWork.DiscreteTimeIntegrator_DSTATE_p <= -3.402823466E+38F) {
        UDC_DWork.DiscreteTimeIntegrator_DSTATE_p = -3.402823466E+38F;
      }
    }
  }

  if (rtb_LogicalOperator_p) {
    UDC_DWork.DiscreteTimeIntegrator_PrevRe_j = 1;
  } else {
    UDC_DWork.DiscreteTimeIntegrator_PrevRe_j = 0;
  }

  /* End of Update for DiscreteIntegrator: '<S112>/Discrete-Time Integrator' */

  /* Update for DiscreteIntegrator: '<S112>/Discrete-Time Integrator1' */
  UDC_DWork.DiscreteTimeIntegrator1_IC_LOAD = 0U;
  if (!rtb_LogicalOperator_p) {
    UDC_DWork.DiscreteTimeIntegrator1_DSTATE += 0.1F * rtb_Product3;
    if (UDC_DWork.DiscreteTimeIntegrator1_DSTATE >= 3.402823466E+38F) {
      UDC_DWork.DiscreteTimeIntegrator1_DSTATE = 3.402823466E+38F;
    } else {
      if (UDC_DWork.DiscreteTimeIntegrator1_DSTATE <= -3.402823466E+38F) {
        UDC_DWork.DiscreteTimeIntegrator1_DSTATE = -3.402823466E+38F;
      }
    }
  }

  if (rtb_LogicalOperator_p) {
    UDC_DWork.DiscreteTimeIntegrator1_PrevRes = 1;
  } else {
    UDC_DWork.DiscreteTimeIntegrator1_PrevRes = 0;
  }

  /* End of Update for DiscreteIntegrator: '<S112>/Discrete-Time Integrator1' */

  /* Update for UnitDelay: '<S8>/Unit Delay' */
  UDC_DWork.UnitDelay_DSTATE_g = rtb_Switch2_h;

  /* Update for UnitDelay: '<S65>/Unit Delay4' */
  UDC_DWork.UnitDelay4_DSTATE_j = UDC_B.TP.LogicalOperator1;

  /* Update for UnitDelay: '<S7>/Unit Delay' */
  UDC_DWork.UnitDelay_DSTATE_c = 108U;
}

/* Model initialize function */
void UDC_initialize(struct fUDC* inst)
{
  /* Registration code */

  /* initialize non-finites */
  rt_InitInfAndNaN(sizeof(real_T));

  /* InitializeConditions for IfAction SubSystem: '<S6>/UrValCntr' */
  /* InitializeConditions for DiscreteIntegrator: '<S94>/Discrete-Time Integrator' */
  UDC_DWork.DiscreteTimeIntegrator_IC_LOA_f = 1U;

  /* InitializeConditions for DiscreteIntegrator: '<S94>/Discrete-Time Integrator1' */
  UDC_DWork.DiscreteTimeIntegrator1_IC_LO_i = 1U;

  /* InitializeConditions for Atomic SubSystem: '<S97>/Filter_DPr' */
  UDC_Filter_Init(&UDC_DWork.Filter_DPr, inst);

  /* End of InitializeConditions for SubSystem: '<S97>/Filter_DPr' */

  /* InitializeConditions for Atomic SubSystem: '<S98>/Filter_DPr' */
  UDC_Filter_Init(&UDC_DWork.Filter_DPr_h, inst);

  /* End of InitializeConditions for SubSystem: '<S98>/Filter_DPr' */

  /* End of InitializeConditions for SubSystem: '<S6>/UrValCntr' */

  /* InitializeConditions for IfAction SubSystem: '<S6>/UrPumpCntr' */
  /* InitializeConditions for DiscreteIntegrator: '<S88>/Discrete-Time Integrator' */
  UDC_DWork.DiscreteTimeIntegrator_IC_LOA_e = 1U;

  /* InitializeConditions for DiscreteIntegrator: '<S88>/Discrete-Time Integrator1' */
  UDC_DWork.DiscreteTimeIntegrator1_IC_LO_n = 1U;

  /* End of InitializeConditions for SubSystem: '<S6>/UrPumpCntr' */
  UDC_PrevZCSigState.Delay_Reset_ZCE = UNINITIALIZED_ZCSIG;
  UDC_PrevZCSigState.Delay_Reset_ZCE_n = UNINITIALIZED_ZCSIG;
  UDC_PrevZCSigState.Delay_Reset_ZCE_d = UNINITIALIZED_ZCSIG;
  UDC_PrevZCSigState.Delay_Reset_ZCE_i = UNINITIALIZED_ZCSIG;
  UDC_PrevZCSigState.Delay_Reset_ZCE_b = UNINITIALIZED_ZCSIG;

  /* InitializeConditions for Atomic SubSystem: '<S9>/E21_NOxCatOutManager' */

  /* InitializeConditions for Atomic SubSystem: '<S119>/TOF' */
  UDC_TOF_Init(&UDC_DWork.TOF, inst);

  /* End of InitializeConditions for SubSystem: '<S119>/TOF' */

  /* InitializeConditions for Atomic SubSystem: '<S119>/TOF1' */
  UDC_TOF_Init(&UDC_DWork.TOF1, inst);

  /* End of InitializeConditions for SubSystem: '<S119>/TOF1' */

  /* End of InitializeConditions for SubSystem: '<S9>/E21_NOxCatOutManager' */

  /* InitializeConditions for Atomic SubSystem: '<S120>/Filter' */
  UDC_Filter_Init(&UDC_DWork.Filter, inst);

  /* End of InitializeConditions for SubSystem: '<S120>/Filter' */

  /* InitializeConditions for Atomic SubSystem: '<S120>/Filter2' */
  UDC_Filter_Init(&UDC_DWork.Filter2, inst);

  /* End of InitializeConditions for SubSystem: '<S120>/Filter2' */

  /* InitializeConditions for Delay: '<S66>/Delay' */
  UDC_DWork.icLoad = 1U;

  /* InitializeConditions for Atomic SubSystem: '<Root>/SlipDetection' */
  /* InitializeConditions for Atomic SubSystem: '<S137>/TOF' */
  /* InitializeConditions for UnitDelay: '<S143>/Unit Delay' */
  UDC_DWork.UnitDelay_DSTATE_jw = TRUE;

  /* InitializeConditions for Delay: '<S147>/Delay' */
  UDC_DWork.icLoad_d = 1U;

  /* End of InitializeConditions for SubSystem: '<S137>/TOF' */

  /* InitializeConditions for Atomic SubSystem: '<S137>/TP' */
  UDC_TP_Init(&UDC_DWork.TP_e, inst);

  /* End of InitializeConditions for SubSystem: '<S137>/TP' */

  /* InitializeConditions for Atomic SubSystem: '<S138>/TP1' */
  UDC_TP_Init(&UDC_DWork.TP1, inst);

  /* End of InitializeConditions for SubSystem: '<S138>/TP1' */

  /* InitializeConditions for Atomic SubSystem: '<S139>/TP' */
  UDC_TP_Init(&UDC_DWork.TP_m, inst);

  /* End of InitializeConditions for SubSystem: '<S139>/TP' */

  /* InitializeConditions for Atomic SubSystem: '<S139>/Filter_OxiIn' */
  UDC_Filter_Init(&UDC_DWork.Filter_OxiIn, inst);

  /* End of InitializeConditions for SubSystem: '<S139>/Filter_OxiIn' */

  /* InitializeConditions for Atomic SubSystem: '<S139>/Filter_CatOut' */
  UDC_Filter_Init(&UDC_DWork.Filter_CatOut, inst);

  /* End of InitializeConditions for SubSystem: '<S139>/Filter_CatOut' */

  /* InitializeConditions for Delay: '<S202>/Delay' */
  UDC_DWork.icLoad_g = 1U;

  /* InitializeConditions for Delay: '<S203>/Delay' */
  UDC_DWork.icLoad_e = 1U;

  /* InitializeConditions for MATLAB Function: '<S141>/switchHold fct1' */
  UDC_DWork.x = TRUE;

  /* End of InitializeConditions for SubSystem: '<Root>/SlipDetection' */

  /* InitializeConditions for Atomic SubSystem: '<S30>/Cell1' */
  UDC_Cell1_Init(&UDC_DWork.Cell1, inst);

  /* End of InitializeConditions for SubSystem: '<S30>/Cell1' */

  /* InitializeConditions for Atomic SubSystem: '<S30>/Cell2' */
  UDC_Cell1_Init(&UDC_DWork.Cell2, inst);

  /* End of InitializeConditions for SubSystem: '<S30>/Cell2' */

  /* InitializeConditions for Atomic SubSystem: '<S30>/Cell3' */
  UDC_Cell1_Init(&UDC_DWork.Cell3, inst);

  /* End of InitializeConditions for SubSystem: '<S30>/Cell3' */

  /* InitializeConditions for DiscreteIntegrator: '<S112>/Discrete-Time Integrator' */
  UDC_DWork.DiscreteTimeIntegrator_IC_LOADI = 1U;

  /* InitializeConditions for DiscreteIntegrator: '<S112>/Discrete-Time Integrator1' */
  UDC_DWork.DiscreteTimeIntegrator1_IC_LOAD = 1U;

  /* InitializeConditions for Atomic SubSystem: '<S15>/Filter' */
  UDC_Filter_Init(&UDC_DWork.Filter_o, inst);

  /* End of InitializeConditions for SubSystem: '<S15>/Filter' */

  /* InitializeConditions for Atomic SubSystem: '<S15>/Filter1' */
  UDC_Filter_Init(&UDC_DWork.Filter1, inst);

  /* End of InitializeConditions for SubSystem: '<S15>/Filter1' */

  /* InitializeConditions for Atomic SubSystem: '<S65>/TP' */
  UDC_TP_Init(&UDC_DWork.TP, inst);

  /* End of InitializeConditions for SubSystem: '<S65>/TP' */
}

/* Model terminate function */
void UDC_terminate(struct fUDC* inst)
{
  /* (no terminate code required) */
}

/*======================== TOOL VERSION INFORMATION ==========================*
 * MATLAB 8.0 (R2012b)20-Jul-2012                                             *
 * Simulink 8.0 (R2012b)20-Jul-2012                                           *
 * Simulink Coder 8.3 (R2012b)20-Jul-2012                                     *
 * Embedded Coder 6.3 (R2012b)20-Jul-2012                                     *
 * Stateflow 8.0 (R2012b)20-Jul-2012                                          *
 *============================================================================*/

/*======================= LICENSE IN USE INFORMATION =========================*
 * matlab                                                                     *
 * matlab_coder                                                               *
 * real-time_workshop                                                         *
 * rtw_embedded_coder                                                         *
 * simulink                                                                   *
 *============================================================================*/
```

#### UDC_data.c
```c
/********************************************************************
 * COPYRIGHT -- Bernecker + Rainer Industrie-Elektronik Ges.m.b.H.
 ********************************************************************
 * Program: UDC
 * File: UDC_data.c
 * Author: 105055527
 * Created: Thu Mar 02 16:51:06 2017
 ********************************************************************
 * Data for program UDC
 ********************************************************************
 * Generated with B&R Automation Studio Target for Simulink V4.2
 * (ERT based)
 ********************************************************************/
#include "UDC.h"
#include "UDC_private.h"

/*  GLOBAL DATA DEFINITIONS */

/* Invariant block signals (auto storage) */
const ConstBlockIO_UDC UDC_ConstB = {
  /* Start of '<S139>/Filter_OxiIn' */
  {
    2.22044605E-16F
    /* '<S179>/Conversion' */
  }
  /* End of '<S139>/Filter_OxiIn' */
  ,

  /* Start of '<S139>/Filter_CatOut' */
  {
    2.22044605E-16F
    /* '<S177>/Conversion' */
  }
  /* End of '<S139>/Filter_CatOut' */
  ,

  /* Start of '<S120>/Filter2' */
  {
    2.22044605E-16F
    /* '<S134>/Conversion' */
  }
  /* End of '<S120>/Filter2' */
  ,

  /* Start of '<S120>/Filter' */
  {
    2.22044605E-16F
    /* '<S132>/Conversion' */
  }
  /* End of '<S120>/Filter' */
  ,

  /* Start of '<S98>/Filter_DPr' */
  {
    2.22044605E-16F
    /* '<S109>/Conversion' */
  }
  /* End of '<S98>/Filter_DPr' */
  ,

  /* Start of '<S97>/Filter_DPr' */
  {
    2.22044605E-16F
    /* '<S104>/Conversion' */
  }
  /* End of '<S97>/Filter_DPr' */
  ,

  /* Start of '<S15>/Filter1' */
  {
    2.22044605E-16F
    /* '<S71>/Conversion' */
  }
  /* End of '<S15>/Filter1' */
  ,

  /* Start of '<S15>/Filter' */
  {
    2.22044605E-16F
    /* '<S69>/Conversion' */
  }
  /* End of '<S15>/Filter' */
};

/* Constant parameters (auto storage) */
const ConstParam_UDC UDC_ConstP = {
  /* Expression: [0 0.3 0.5 0.75 1]
   * Referenced by: '<S12>/Constant'
   */
  { 0.0, 0.3, 0.5, 0.75, 1.0 },

  /* Computed Parameter: InterpolationUsingPre
   * Referenced by: '<S59>/Interpolation Using Prelookup'
   */
  { 2U, 5U },

  /* Pooled Parameter (Expression: [0 1;1 0;0 1;0 1;1 0;1 0;0 0;0 0])
   * Referenced by:
   *   '<S156>/Logic'
   *   '<S200>/Logic'
   */
  { 0, 1, 0, 0, 1, 1, 0, 0, 1, 0, 1, 1, 0, 0, 0, 0 }
};
```

#### fUDC.c
```c
/********************************************************************
 * COPYRIGHT -- Bernecker + Rainer Industrie-Elektronik Ges.m.b.H.
 ********************************************************************
 * Program: UDC
 * File: fUDC.c
 * Author: 105055527
 * Created: Thu Mar 02 16:51:06 2017
 ********************************************************************
 * Implementation of program UDC
 ********************************************************************
 * Generated with B&R Automation Studio Target for Simulink V4.2
 * (ERT based)
 ********************************************************************/
#include <bur/plctypes.h>
#include "UDC.h"
#include "rtwtypes.h"

/* Defines */
#define SS_TERMINATE 4
#define SS_OUTPUT 3
#define SS_INITIALIZE 2

/*  Data Types */

/**************************** GLOBAL DATA *************************************/
/*  Definitions */

/*  Declarations  */

/***************************** FILE SCOPE DATA ********************************/

/*************************** FUNCTIONS ****************************************/
#ifdef __cplusplus

unsigned long bur_heap_size = 6553500;

#endif

void fUDC(struct fUDC* inst)
{

  switch (inst->ssMethodType)
  {
   case SS_INITIALIZE:
    /* call model initialize function */
    UDC_initialize(inst);
    break;

   case SS_OUTPUT:
    /* call model step function */
    UDC_step(inst);

    break;

   case SS_TERMINATE:
    /* call model terminate function */
    UDC_terminate(inst);
    break;
  }
}

/*****************************************************************************
   Function block sample time: 0.099999999999999992s
 *****************************************************************************/

/*****************************************************************************
   B&R Automation Studio Target for Simulink Version: A4.5.1 (27-Jul-2015)
 *****************************************************************************/

/*======================== TOOL VERSION INFORMATION ==========================*
 * MATLAB 8.0 (R2012b)20-Jul-2012                                             *
 * Simulink 8.0 (R2012b)20-Jul-2012                                           *
 * Simulink Coder 8.3 (R2012b)20-Jul-2012                                     *
 * Embedded Coder 6.3 (R2012b)20-Jul-2012                                     *
 * Stateflow 8.0 (R2012b)20-Jul-2012                                          *
 *============================================================================*/

/*======================= LICENSE IN USE INFORMATION =========================*
 * matlab                                                                     *
 * matlab_coder                                                               *
 * real-time_workshop                                                         *
 * rtw_embedded_coder                                                         *
 * simulink                                                                   *
 *============================================================================*/
```

#### rtGetInf.c
```c
/********************************************************************
 * COPYRIGHT -- Bernecker + Rainer Industrie-Elektronik Ges.m.b.H.
 ********************************************************************
 * Program: UDC
 * File: rtGetInf.c
 * Author: 105055527
 * Created: Thu Mar 02 16:51:06 2017
 ********************************************************************
 * Implementation of program UDC
 ********************************************************************
 * Generated with B&R Automation Studio Target for Simulink V4.2
 * (ERT based)
 ********************************************************************/
/*
 * Abstract:
 *      Function to intialize non-finite, Inf
 */

#include "rtGetInf.h"

/*  Defines */
#define NumBitsPerChar                 8U

/*  Data Types */

/**************************** GLOBAL DATA *************************************/
/*  Definitions */

/*  Declarations  */

/***************************** FILE SCOPE DATA ********************************/

/*************************** FUNCTIONS ****************************************/

/*
 * Initialize rtInf needed by the generated code.
 * Inf is initialized as non-signaling. Assumes IEEE.
 */
real_T rtGetInf(void)
{
  size_t bitsPerReal = sizeof(real_T) * (NumBitsPerChar);
  real_T inf = 0.0;
  if (bitsPerReal == 32U) {
    inf = rtGetInfF();
  } else {
    union {
      LittleEndianIEEEDouble bitVal;
      real_T fltVal;
    } tmpVal;

    tmpVal.bitVal.words.wordH = 0x7FF00000U;
    tmpVal.bitVal.words.wordL = 0x00000000U;
    inf = tmpVal.fltVal;
  }

  return inf;
}

/*
 * Initialize rtInfF needed by the generated code.
 * Inf is initialized as non-signaling. Assumes IEEE.
 */
real32_T rtGetInfF(void)
{
  IEEESingle infF;
  infF.wordL.wordLuint = 0x7F800000U;
  return infF.wordL.wordLreal;
}

/*
 * Initialize rtMinusInf needed by the generated code.
 * Inf is initialized as non-signaling. Assumes IEEE.
 */
real_T rtGetMinusInf(void)
{
  size_t bitsPerReal = sizeof(real_T) * (NumBitsPerChar);
  real_T minf = 0.0;
  if (bitsPerReal == 32U) {
    minf = rtGetMinusInfF();
  } else {
    union {
      LittleEndianIEEEDouble bitVal;
      real_T fltVal;
    } tmpVal;

    tmpVal.bitVal.words.wordH = 0xFFF00000U;
    tmpVal.bitVal.words.wordL = 0x00000000U;
    minf = tmpVal.fltVal;
  }

  return minf;
}

/*
 * Initialize rtMinusInfF needed by the generated code.
 * Inf is initialized as non-signaling. Assumes IEEE.
 */
real32_T rtGetMinusInfF(void)
{
  IEEESingle minfF;
  minfF.wordL.wordLuint = 0xFF800000U;
  return minfF.wordL.wordLreal;
}

/*======================== TOOL VERSION INFORMATION ==========================*
 * MATLAB 8.0 (R2012b)20-Jul-2012                                             *
 * Simulink 8.0 (R2012b)20-Jul-2012                                           *
 * Simulink Coder 8.3 (R2012b)20-Jul-2012                                     *
 * Embedded Coder 6.3 (R2012b)20-Jul-2012                                     *
 * Stateflow 8.0 (R2012b)20-Jul-2012                                          *
 *============================================================================*/

/*======================= LICENSE IN USE INFORMATION =========================*
 * matlab                                                                     *
 * matlab_coder                                                               *
 * real-time_workshop                                                         *
 * rtw_embedded_coder                                                         *
 * simulink                                                                   *
 *============================================================================*/
```

#### rtGetNaN.c
```c
/********************************************************************
 * COPYRIGHT -- Bernecker + Rainer Industrie-Elektronik Ges.m.b.H.
 ********************************************************************
 * Program: UDC
 * File: rtGetNaN.c
 * Author: 105055527
 * Created: Thu Mar 02 16:51:06 2017
 ********************************************************************
 * Implementation of program UDC
 ********************************************************************
 * Generated with B&R Automation Studio Target for Simulink V4.2
 * (ERT based)
 ********************************************************************/
/*
 * Abstract:
 *      Function to intialize non-finite, NaN
 */

#include "rtGetNaN.h"

/*  Defines */
#define NumBitsPerChar                 8U

/*  Data Types */

/**************************** GLOBAL DATA *************************************/
/*  Definitions */

/*  Declarations  */

/***************************** FILE SCOPE DATA ********************************/

/*************************** FUNCTIONS ****************************************/

/*
 * Initialize rtNaN needed by the generated code.
 * NaN is initialized as non-signaling. Assumes IEEE.
 */
real_T rtGetNaN(void)
{
  size_t bitsPerReal = sizeof(real_T) * (NumBitsPerChar);
  real_T nan = 0.0;
  if (bitsPerReal == 32U) {
    nan = rtGetNaNF();
  } else {
    union {
      LittleEndianIEEEDouble bitVal;
      real_T fltVal;
    } tmpVal;

    tmpVal.bitVal.words.wordH = 0xFFF80000U;
    tmpVal.bitVal.words.wordL = 0x00000000U;
    nan = tmpVal.fltVal;
  }

  return nan;
}

/*
 * Initialize rtNaNF needed by the generated code.
 * NaN is initialized as non-signaling. Assumes IEEE.
 */
real32_T rtGetNaNF(void)
{
  IEEESingle nanF = { { 0 } };

  nanF.wordL.wordLuint = 0xFFC00000U;
  return nanF.wordL.wordLreal;
}

/*======================== TOOL VERSION INFORMATION ==========================*
 * MATLAB 8.0 (R2012b)20-Jul-2012                                             *
 * Simulink 8.0 (R2012b)20-Jul-2012                                           *
 * Simulink Coder 8.3 (R2012b)20-Jul-2012                                     *
 * Embedded Coder 6.3 (R2012b)20-Jul-2012                                     *
 * Stateflow 8.0 (R2012b)20-Jul-2012                                          *
 *============================================================================*/

/*======================= LICENSE IN USE INFORMATION =========================*
 * matlab                                                                     *
 * matlab_coder                                                               *
 * real-time_workshop                                                         *
 * rtw_embedded_coder                                                         *
 * simulink                                                                   *
 *============================================================================*/
```

#### rt_nonfinite.c
```c
/********************************************************************
 * COPYRIGHT -- Bernecker + Rainer Industrie-Elektronik Ges.m.b.H.
 ********************************************************************
 * Program: UDC
 * File: rt_nonfinite.c
 * Author: 105055527
 * Created: Thu Mar 02 16:51:06 2017
 ********************************************************************
 * Implementation of program UDC
 ********************************************************************
 * Generated with B&R Automation Studio Target for Simulink V4.2
 * (ERT based)
 ********************************************************************/
/*
 * Abstract:
 *      Function to intialize non-finites,
 *      (Inf, NaN and -Inf).
 */

#include "rt_nonfinite.h"
#include "rtGetNaN.h"
#include "rtGetInf.h"

/*  Defines */

/*  Data Types */

/**************************** GLOBAL DATA *************************************/
/*  Definitions */

/*  Declarations  */
real_T rtInf;
real_T rtMinusInf;
real_T rtNaN;
real32_T rtInfF;
real32_T rtMinusInfF;
real32_T rtNaNF;

/***************************** FILE SCOPE DATA ********************************/

/*************************** FUNCTIONS ****************************************/

/*
 * Initialize the rtInf, rtMinusInf, and rtNaN needed by the
 * generated code. NaN is initialized as non-signaling. Assumes IEEE.
 */
void rt_InitInfAndNaN(size_t realSize)
{
  (void) (realSize);
  rtNaN = rtGetNaN();
  rtNaNF = rtGetNaNF();
  rtInf = rtGetInf();
  rtInfF = rtGetInfF();
  rtMinusInf = rtGetMinusInf();
  rtMinusInfF = rtGetMinusInfF();
}

/* Test if value is infinite */
boolean_T rtIsInf(real_T value)
{
  return (boolean_T)((value==rtInf || value==rtMinusInf) ? 1U : 0U);
}

/* Test if single-precision value is infinite */
boolean_T rtIsInfF(real32_T value)
{
  return (boolean_T)(((value)==rtInfF || (value)==rtMinusInfF) ? 1U : 0U);
}

/* Test if value is not a number */
boolean_T rtIsNaN(real_T value)
{
  return (boolean_T)((value!=value) ? 1U : 0U);
}

/* Test if single-precision value is not a number */
boolean_T rtIsNaNF(real32_T value)
{
  return (boolean_T)(((value!=value) ? 1U : 0U));
}

/*======================== TOOL VERSION INFORMATION ==========================*
 * MATLAB 8.0 (R2012b)20-Jul-2012                                             *
 * Simulink 8.0 (R2012b)20-Jul-2012                                           *
 * Simulink Coder 8.3 (R2012b)20-Jul-2012                                     *
 * Embedded Coder 6.3 (R2012b)20-Jul-2012                                     *
 * Stateflow 8.0 (R2012b)20-Jul-2012                                          *
 *============================================================================*/

/*======================= LICENSE IN USE INFORMATION =========================*
 * matlab                                                                     *
 * matlab_coder                                                               *
 * real-time_workshop                                                         *
 * rtw_embedded_coder                                                         *
 * simulink                                                                   *
 *============================================================================*/
```

#### lib_properties.txt
```
For manual assignment to hardware configuration please
add the following additional include directories:

\Logical\MATLAB_includes\R2012b\

And the following additional build options:

-lm -D MODEL=UDC -D NUMST=1 -D NCSTATES=0 -D HAVESTDIO -D ONESTEPFCN=1 -D TERMFCN=1 -D MAT_FILE=0 -D MULTI_INSTANCE_CODE=0 -D INTEGER_CODE=0 -D MT=0 -D CLASSIC_INTERFACE=0 -D TID01EQ=0
```

### Data object Logical/Emission/META_EM (Simple) - MODUL META data file

#### META_EM.dat
```
; *******************************************************************************
; AGGR: Module Meta Data (data module)
;
; This code is confidential and proprietary to the INNIO Company.
; It may not be used in any form, or reproduced in any manner, without the express
; written permission of the INNIO Company.
; Copyright, INNIO Company, 2023
;
; Customized modifications: -
; ------------------------
;
; History:
; -------
; V3.99		06-03-2013	Weitzer, generated for modular software
; 	 		17-07-2013	Zengerer, Strukturupdate
;       	04-12.2013  Maxhera, content update
; V4.00 	31.01.2014	Weitzer, versions changed
; V4.03 	09-03-2016	Mari W., adaption after adding SCR CAT
;						Weitzer, corrections
; V4.04 	07-11-2016	Weitzer, MM2VIS.rNOx_NOxS_EngOut_mg & MM2VIS.rNOx_NOxS_CatOut_mg added
; V4.05		17-05-2017	Messner, move SCR to EM module
;						Tinello, SCR update to Spec version a
;								 NOx sensor integrated
; V4.05.03	13-02-2018	Tinello, Mittelwert-Berechnung korrigiert, dosing stop, sample gas pump and emission monitoring changed
;								 Dependencies angepasst
; V4.05.04	19-03-2018	Tinello, NOx sensor task angepasst / Para Check erweitert
; V4.05.05	23-05-2018	Tinello, Bugfix SCR
; V4.05.06	20-09-2018	Tinello, Bugfix SCR, NOx -> bu
; V4.06.00	16-03-2018	Hohens., ".Exist" added to HALioBase library for analog inputs --> fixed type casting in SCR_UDC
; V4.07.00	11-04-2019	Tinello, NOx: bugfix; plausibility check for O2 and NOx, deviation bank A/B, status overview added
;								 SCR: Length of urea dosing line, new warning for dosing error, Urea pump stop – overpressure,
;									  manual mode only 30m, MSS always active
;								 EM:  Average calculation and monitoring moved from SCR to Emission task
; V4.07.01	06-11-2019	Tinello, NOx: new lifetime parameter; plausibility check changed; O2-filter for conversion of NOx setpoint added; reduced perm file write interval (bu1)
; V4.09.00	04-03-2020	Tinello, plausibility and self-diagnosis changed -> Spec. (c)
; V4.09.02	31.08.2020	Tinello, (=BU2) bugfix -> Message 2455 only active if urea dosing controller is active / CAN read operating hours / CEMS correction
; V4.10.00	28.01.2021	Tinello, BugFix: Timer & other FuB's / Sum emission error extended / urea supply pump starts earlier
;			15.06.2021	Tinello, BU02: Operating Hours NOx / unteres O2-Limit von 5% -> 0% / DailyAvg -> perm
; V4.11.00	29.03.2022	Tinello, Interpolation of load dependent NOx-setpoint / BugFix: NOx plausibility check changed: Skip-mode considered / SCR bugfixes / CAT temp min monitoring
; 			03.08.2022	Tinello, BU01: NOx sensor activation independent of temperature after 5min/10min of start speed
; V4.12.00	14.11.2022	Arnold,  H2 based EngOut NOx setpoint for UDC
;			30.01.2023	Tinello	 SCR Customer added
; V4.13.00	20.11.2023	Farre,	 Replaced Para.rP_Set_Min_Norm by IN_GR.rP_Set_Min_Norm interface coming from OP. (2023-168)
; 			21.11.2023	Tinello, Added urea tank level, new warnings and operational messages, release dosing & slip detection adapted / W3456 split (2022-141)
;								 Temp changed for NOx sensor start (2023-191)
; V4.14.00	18.06.2024	Soto,	 Low NOx sensor with CAN communication (2023-183)
;			21.10.2024	Farre,	 CEMS internal modifications (2023-183)
;			25.11.2024	Bacci,	 T6 Start procedure with purge start (2024-219): effect of elimination of scavenging fan on sensors calibration
;
; Instructions for use:
; --------------------
; make only changes at the version numbers
; OBEY XML FORMATING RULES!
;
; Outstandings:
; ------------
;
; *******************************************************************************
;
"<META>"
;
; Module ID
"<MODUL>EM</MODUL>"
;
; Module Version (xx.yy.zz.cc)
"<VERSION>04.14.00.00</VERSION>"
;
; Module Basisupdate Version BU (00-99)
"<BASISUPDATE_VERSION>00</BASISUPDATE_VERSION>"
;
; Optional: specify order number for limitated module usage
"<ORDER></ORDER>" ;<!--(optional for restricted customizations; missing statement makes module valid for all orders)-->
;
; Parameter Check <PARAn Name='aAbcdef' MIN='xxx' MAX='yyy' />  (watch for correct spacings and apostrophs!)
"<PARAMETER_CHK>"
"<PARA1 Name='rN_EngStart_LimHi' MIN='50.0' MAX='2200.0' />"
"<PARA2 Name='iEng_Motortype' MIN='208' MAX='920' />"
"<PARA3 />"
"<PARA4 />"
"<PARA5 />"
"</PARAMETER_CHK>"
;
; Permanent Datamodule Filenames<!-- NAME ist ohne Dateiendung einzutragen; Nur für Counter und interne Parameter verwenden-->
"<DATAMODULES>" ;<!-- optional; mehrere DATAMODULES erlaubt-->
"	<DATAMODULE>par_EM</DATAMODULE>"
"	<DATAMODULE>perm_EM</DATAMODULE>"
"</DATAMODULES>"
;
; Dependencies Modules (MMxx.yy.zz.cc)
"<DEPENDENCIES>"
"	<DEPENDENCY MODULE='AB' VERSION='04.00.00.00' />"
"	<DEPENDENCY MODULE='AG' VERSION='04.00.00.00' />"
"	<DEPENDENCY MODULE='CH' VERSION='04.05.00.00' />"
"	<DEPENDENCY MODULE='CP' VERSION='04.05.00.00' />"
"	<DEPENDENCY MODULE='EC' VERSION='04.12.00.00' />"
"	<DEPENDENCY MODULE='EG' VERSION='04.00.00.00' />"
"	<DEPENDENCY MODULE='EX' VERSION='04.05.00.00' />"
"	<DEPENDENCY MODULE='HA' VERSION='04.14.00.00' />"
"	<DEPENDENCY MODULE='IG' VERSION='04.00.00.00' />"
"	<DEPENDENCY MODULE='OP' VERSION='04.13.00.00' />"
"	<DEPENDENCY MODULE='PB' VERSION='04.06.00.00' />"
"   <DEPENDENCY VISVERSION='02.15.00.00' />"				;Dependencies Visualization
"</DEPENDENCIES>"
;
; Module function description
"<MODULEFUNCTION>" ;<!-- short overview documentation of module function; add reference to detailed information, if available-->
"	<General>	"
"	measure NOx and O2 with NOx sensor "
"	</General>	"
""
"	<F1 Name='measure NOx and O2' LastModified='04.00.00.00'>"
"	initiate CAN communication, measure NOx and O2 value	"
"	</F1>"
"	<F2 Name=' alarm management' LastModified='04.00.00.00'>"
"   Message for Emission "
"	</F2>"
"	<F3 Name=' alarm management' LastModified='04.05.06.00'>"
"   SCR included / NOx included"
"	NOx monitoring and availability of signals 180s after sensor start"
"	SCR Adjustment with ext CEMS"
"	</F3>"
"	<F4 Name=' emission monitoring' LastModified='04.07.00.00'>"
"	NOx sensor self diagnosis, plausibility check, deviation bank A/B and status overview added"
"	MsErr now also active with operation mode selector switch in OFF mode"
"	2 DI's for external SCR systems, length of urea dosing line and new warning for dosing error added"
"	Transformation from mg/Nm3 --> ppm and ppm --> mg/Nm3 added"
"	Average calculation and monitoring adapted to new spec (Daily average calculation for NOx added. Emission monitoring with limit and tolerance)"
"	Counter for Duration of emission tolerance exceedance added"
"	</F4>"
"	<F5 Name=' emission monitoring' LastModified='04.07.01.00'>"
"	reduced perm file write interval to avoid CF card wear down"
"	new lifetime parameter; plausibility check changed; O2-filter for conversion of NOx setpoint parameter added"
"	</F5>"
"	<F6 Name=' emission monitoring' LastModified='04.09.00.00'>"
"	plausibility check changed for CAT out sensor / self-diagnosis 900s after engine shutdown, if CAT out sensor is requested"
"	If during self-diagnosis the result is not available -> try again 3 times before exit self-diagnosis -> Spec. (c)"
"	Release of emission average monitoring changed"
"	</F6>"
"	<F7 Name='CEMS/NOx reading' LastModified='04.09.02.00 BU2'>"
"	bugfix -> Message 2455 only active if urea dosing controller is active"
"	bugfix -> reading operating hours via CAN"
"	bugfix -> CEMS correction only during active NOx sensor"
"	</F7>"
"	<F8 Name='BugFix' LastModified='04.10.00.00'>"
"	BugFix: Timer & other FuB's / Sum emission error extended / urea supply pump starts earlier"
"	</F8>"
"	<F9 Name='BugFix' LastModified='04.10.00.00 BU2'>"
"	BugFix: Operating Hours NOx / unteres O2-Limit von 5% -> 0% / Save daily average permanent"
"	</F9>"
"	<F10 Name='BugFix' LastModified='04.11.00.00'>"
"	Interpolation of load dependent NOx-setpoint"
"	3 new parameters"
"	NOx plausibility check changed: Skip-mode considered"
"	SCR leakage monitoring extended and time changed from 60s ->300s / urea dosing pump - error corrected"
"	Monitoring of CAT-temperature minimum added"
"	BugFix of emission short term average monitoring"
"	</F10>"
"	<F11 Name='BugFix' LastModified='04.11.00.00 BU1'>"
"	Take CO and NOx values from SCR already if limits reached / O2-limit for NOx-Transformation to mg added"
"	Release NOx average monitoring for SCR latest if 20min minimum power reached"
"	SCR temperature difference monitoring changed from 100C to 20C"
"	NOx sensor activation independent of temperature / restart of sensor not before 1s of no connection"
"	</F11>"
"	<F12 Name='SCR features' LastModified='04.13.00.00'>"
"	Added urea tank level, new warnings and operational messages, release dosing & slip detection adapted / W3456 split"
"	Temp changed for NOx sensor start"
"	</F12>"
""
"	<Info>"
"	no furhter information	"
"	</Info>"
""
"	<Customized LastModified='04.00.00.00'>	"
"	- Nothing "
"	</Customized>	"
""
"</MODULEFUNCTION>"
;
"</META>"
```
